# B&R Automation Studio project ControlPLC_DataDistribution
Automation Studio 4.11.3.51 SP; VulcanForms Printer Control PLC Gen 3.0; technology packages: mapp 5.19.0, mappCockpit 5.19.0, mappControl 5.19.0, mappMotion 5.19.3, mappSafety 5.19.0, mappView 5.19.0

## Configuration APC910

CPU 5PC900.TS17-02, AutomationRuntime D4.92, Build 4.1.2, Vc V4.72.5

### Hardware
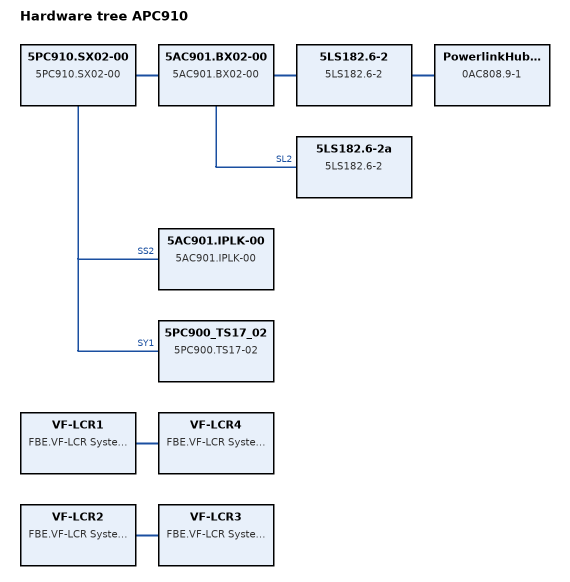
```
5AC901.BX02-00 : 5AC901.BX02-00 v1.0.1.0  [SY -> 5PC910.SX02-00.SY3]
5AC901.IPLK-00 : 5AC901.IPLK-00 v1.8.1.0  [SS -> 5PC910.SX02-00.SS2]
  Supervision = off
5LS182.6-2 : 5LS182.6-2 v1.9.0.0  [SL -> 5AC901.BX02-00.SL1]
  Connector IF1:
    CycleTime = 800
    EplNatSubnet = 192.168.102.0
  Supervision = off
5LS182.6-2a : 5LS182.6-2 v1.9.0.0  [SL -> 5AC901.BX02-00.SL2]
  Connector IF1:
    EplNatSubnet = 192.168.103.0
  Supervision = off
5PC900_TS17_02 : 5PC900.TS17-02 v2.1.0.0  [SY -> 5PC910.SX02-00.SY1]
  ConfigurationID = ControlPLC_LaserCleanroom_APC910
  UserPartitionSize = 5000
  UserRamDevice = PCI.2.LS182.SRAM
  UserRamSize = 1048320
  RemMemDevice = PCI.1.LS182.SRAM
  RemMemSize = 116736
  PermanentPvSize = 50000
  RemanentGlobalPvSize = 50000
  VolatileGlobalPvSize = 1100000
  ClearNvMemoryAfterShutdownFlushError = 0
  CyclicFlushRemMemSelector = 1
  RebootReset = 1
  FileDevice1
  FileDeviceName1 = USER
  FileDevicePath1 = USER_PATH
  FtpUser1
  FtpUsername1 = admin
  FtpUserPassword1 = cjYgzx2XKeawARoLvdaLrZty7HtHCNS4hNwff38YIhA=
  FtpUserSalt1 = Vifl6tjb
  FTPAccessRight1 = 0
  FTPdevice1 = ALL
  ActivateOpcUa = 1
  OpcUaPort = 4850
  OpcUa_Security_AdminRole = Administrators
  OpcUaLimitsMaxPublish = 50
  OpcUaInformationModels_PV_Version = 1
5PC910.SX02-00 : 5PC910.SX02-00 v2.1.2.0
  Connector IF1:
    AssignedOperatingSystem = ARemb
  Connector IF3:
    AssignedOperatingSystem = ARemb
    ActivateDevice = 1
    Mode = Manual
    InternetAddress = 192.168.200.50
    SubnetMask = 255.255.255.0
  Connector IF4:
    AssignedOperatingSystem = ARemb
    ActivateDevice = 1
  Connector IF5:
    AssignedOperatingSystem = ARemb
  Connector IF6:
    AssignedOperatingSystem = ARemb
  Connector IF7:
    AssignedOperatingSystem = ARemb
  Connector IF8:
    AssignedOperatingSystem = ARemb
  Connector IF9:
    AssignedOperatingSystem = ARemb
PowerlinkHub_DCEnclosure : 0AC808.9-1 v1.0.0.0  [ETH1 -> 5LS182.6-2.IF1 [Cable Type=PowerlinkCable, Length=10, Version=1.0.0.3]; ETH6 -> VF-LCR4.PLK2 [Cable Type=PowerlinkCable, Length=10, Version=1.0.0.3]]
VF-LCR1 : FBE.VF-LCR System (version 04) v04 (OrderNumber=VF-LCR)  [PLK1 -> VF-LCR2.PLK2 (NodeNumber=51) [Cable Type=PowerlinkCable, Length=10, Version=1.0.0.3]; PLK2 -> VF-LCR4.PLK1 (NodeNumber=51) [Cable Type=PowerlinkCable, Length=10, Version=1.0.0.3]]
  Supervision = off
  ResponseTimeout = 50
VF-LCR2 : FBE.VF-LCR System (version 04) v04 (OrderNumber=VF-LCR)  [PLK1 -> VF-LCR3.PLK2 (NodeNumber=52) [Cable Type=PowerlinkCable, Length=10, Version=1.0.0.3]; PLK2 -> VF-LCR1.PLK1 (NodeNumber=52) [Cable Type=PowerlinkCable, Length=10, Version=1.0.0.3]]
  Supervision = off
  ResponseTimeout = 50
VF-LCR3 : FBE.VF-LCR System (version 04) v04 (OrderNumber=VF-LCR)  [PLK2 -> VF-LCR2.PLK1 (NodeNumber=53) [Cable Type=PowerlinkCable, Length=10, Version=1.0.0.3]]
  Supervision = off
  ResponseTimeout = 50
VF-LCR4 : FBE.VF-LCR System (version 04) v04 (OrderNumber=VF-LCR)  [PLK1 -> VF-LCR1.PLK2 (NodeNumber=54) [Cable Type=PowerlinkCable, Length=10, Version=1.0.0.3]; PLK2 -> PowerlinkHub_DCEnclosure.ETH6 (NodeNumber=54) [Cable Type=PowerlinkCable, Length=10, Version=1.0.0.3]]
  Supervision = off
  ResponseTimeout = 50
```

### IoMap.iom - 5PC900_TS17_02/IoMap.iom
```iecst
VAR_CONFIG
	::VFLCR_Ope1:IO.raw.oSystemControl AT %QD."VF-LCR2".SYSTEM_CONTROL_I2004Out;
	::VFLCR_Ope1:IO.ao.SelectedPrintNumber AT %QD."VF-LCR2".SELECTED_PRINT_NUMBER_I200BOut;
	::VFLCR_Ope1:IO.ao.SelectedLayerNumber AT %QD."VF-LCR2".SELECTED_LAYER_NUMBER_I200COut;
	::VFLCR_Ope1:IO.ao.SelectedBuildLayout AT %QD."VF-LCR2".SELECTED_BUILD_LAYOUT_I200AOut;
	::VFLCR_Ope1:IO.ao.PLCHeartbeat AT %QD."VF-LCR2".PLC_HEARTBEAT_I2003Out;
	::VFLCR_Ope1:IO.raw.oOperationControl AT %QD."VF-LCR2".OPERATION_CONTROL_I2005Out;
	::VFLCR_Ope1:IO.raw.oManualLaserOperation AT %QD."VF-LCR2".MANUAL_LASER_OPERATION_I200EOut;
	::VFLCR_Ope1:IO.raw.oManualLaserCurrentSetpoint AT %QD."VF-LCR2".MANUAL_LASER_CURRENT_SETPOINT_I200FOut;
	::VFLCR_Ope1:IO.raw.oLaserEnable AT %QD."VF-LCR2".LASER_ENABLE_I2008Out;
	::VFLCR_Ope1:IO.raw.oEnableLaserMainPower AT %QD."VF-LCR2".LASER_REMOTE_START_I2010Out;
	::VFLCR_Ope1:IO.raw.oEnableLaserEmission AT %QD."VF-LCR2".LASER_EMISSION_CONTROL_I2012Out;
	::VFLCR_Ope1:IO.raw.oEnableGuideLaser AT %QD."VF-LCR2".GUIDE_LASER_CONTROL_I2011Out;
	::VFLCR_Ope1:IO.raw.oResetLaserErrors AT %QD."VF-LCR2".LASER_RESET_I2013Out;
	::VFLCR_Ope1:IO.di.PowerlinkModuleOK AT %IX."VF-LCR2".ModuleOk;
	::VFLCR_Ope1:IO.ai.DMACurrentTrajectory[0] AT %ID."VF-LCR2".Entry_I201B_S01;
	::VFLCR_Ope1:IO.raw.iLaserFatalError AT %ID."VF-LCR2".SYSTEM_ERROR_I2018;
	::VFLCR_Ope1:IO.raw.iSystemStatus AT %ID."VF-LCR2".SYSTEM_STATUS_I2006;
	::VFLCR_Ope1:IO.ai.SystemHeartbeat AT %ID."VF-LCR2".SYSTEM_HEARTBEAT_I2002;
	::VFLCR_Ope1:IO.raw.iSoftwareRevision AT %ID."VF-LCR2".SOFTWARE_REVISION_I201D;
	::VFLCR_Ope1:IO.raw.iOperationStatus AT %ID."VF-LCR2".OPERATION_STATUS_I2007;
	::VFLCR_Ope1:IO.raw.iManualModeLaserPower AT %ID."VF-LCR2".LASER_POWER_MONITOR_I2019;
	::VFLCR_Ope1:IO.ai.LUTFiles_CalibrationID AT %ID."VF-LCR2".LUT_LOAD_STATUS_I2009;
	::VFLCR_Ope1:IO.raw.iLaserWatchdogError AT %ID."VF-LCR2".LASER_WATCHDOG_ERROR_I201E;
	::VFLCR_Ope1:IO.raw.iLaserEmissionEnabled AT %ID."VF-LCR2".LASER_EMISSION_ON_I2017;
	::VFLCR_Ope1:IO.raw.iLaserControlPowerEnabled AT %ID."VF-LCR2".LASER_CONTROL_SYSTEM_POWERED_ON_I2015;
	::VFLCR_Ope1:IO.raw.iFPGARevision AT %ID."VF-LCR2".FPGA_REVISION_I2001;
	::VFLCR_Ope1:IO.ai.DMAStatus[8] AT %ID."VF-LCR2".Entry_I201A_S09;
	::VFLCR_Ope1:IO.ai.DMAStatus[7] AT %ID."VF-LCR2".Entry_I201A_S08;
	::VFLCR_Ope1:IO.ai.DMAStatus[6] AT %ID."VF-LCR2".Entry_I201A_S07;
	::VFLCR_Ope1:IO.ai.DMAStatus[5] AT %ID."VF-LCR2".Entry_I201A_S06;
	::VFLCR_Ope1:IO.ai.DMAStatus[4] AT %ID."VF-LCR2".Entry_I201A_S05;
	::VFLCR_Ope1:IO.ai.DMAStatus[3] AT %ID."VF-LCR2".Entry_I201A_S04;
	::VFLCR_Ope1:IO.ai.DMAStatus[13] AT %ID."VF-LCR2".Entry_I201A_S0E;
	::VFLCR_Ope1:IO.ai.DMAStatus[2] AT %ID."VF-LCR2".Entry_I201A_S03;
	::VFLCR_Ope1:IO.ai.DMAStatus[19] AT %ID."VF-LCR2".Entry_I201A_S14;
	::VFLCR_Ope1:IO.ai.DMAStatus[1] AT %ID."VF-LCR2".Entry_I201A_S02;
	::VFLCR_Ope1:IO.ai.DMAStatus[18] AT %ID."VF-LCR2".Entry_I201A_S13;
	::VFLCR_Ope1:IO.ai.DMAStatus[17] AT %ID."VF-LCR2".Entry_I201A_S12;
	::VFLCR_Ope1:IO.ai.DMAStatus[16] AT %ID."VF-LCR2".Entry_I201A_S11;
	::VFLCR_Ope1:IO.ai.DMAStatus[15] AT %ID."VF-LCR2".Entry_I201A_S10;
	::VFLCR_Ope1:IO.ai.DMAStatus[14] AT %ID."VF-LCR2".Entry_I201A_S0F;
	::VFLCR_Ope1:IO.raw.iLaserMainPowerEnabled AT %ID."VF-LCR2".LASER_MAIN_POWER_ON_I2016;
	::VFLCR_Ope1:IO.raw.iLaserReady_Error AT %ID."VF-LCR2".LASER_ERROR_READY_I2014;
	::VFLCR_Ope1:IO.ai.DMAStatus[20] AT %ID."VF-LCR2".Entry_I201A_S15;
	::VFLCR_Ope1:IO.ai.DMAStatus[12] AT %ID."VF-LCR2".Entry_I201A_S0D;
	::VFLCR_Ope1:IO.ai.DMACurrentTrajectory[7] AT %ID."VF-LCR2".Entry_I201B_S08;
	::VFLCR_Ope1:IO.ai.DMAStatus[0] AT %ID."VF-LCR2".Entry_I201A_S01;
	::VFLCR_Ope1:IO.ai.DMALastPacketPosition[8] AT %ID."VF-LCR2".Entry_I201C_S09;
	::VFLCR_Ope1:IO.ai.DMALastPacketPosition[7] AT %ID."VF-LCR2".Entry_I201C_S08;
	::VFLCR_Ope1:IO.ai.DMALastPacketPosition[6] AT %ID."VF-LCR2".Entry_I201C_S07;
	::VFLCR_Ope1:IO.ai.DMALastPacketPosition[5] AT %ID."VF-LCR2".Entry_I201C_S06;
	::VFLCR_Ope1:IO.ai.DMALastPacketPosition[4] AT %ID."VF-LCR2".Entry_I201C_S05;
	::VFLCR_Ope1:IO.ai.DMALastPacketPosition[3] AT %ID."VF-LCR2".Entry_I201C_S04;
	::VFLCR_Ope1:IO.ai.DMALastPacketPosition[2] AT %ID."VF-LCR2".Entry_I201C_S03;
	::VFLCR_Ope1:IO.ai.DMALastPacketPosition[19] AT %ID."VF-LCR2".Entry_I201C_S14;
	::VFLCR_Ope1:IO.ai.DMAStatus[9] AT %ID."VF-LCR2".Entry_I201A_S0A;
	::VFLCR_Ope1:IO.ai.DMALastPacketPosition[20] AT %ID."VF-LCR2".Entry_I201C_S15;
	::VFLCR_Ope1:IO.ai.DMALastPacketPosition[18] AT %ID."VF-LCR2".Entry_I201C_S13;
	::VFLCR_Ope1:IO.ai.DMALastPacketPosition[17] AT %ID."VF-LCR2".Entry_I201C_S12;
	::VFLCR_Ope1:IO.ai.DMALastPacketPosition[16] AT %ID."VF-LCR2".Entry_I201C_S11;
	::VFLCR_Ope1:IO.ai.DMALastPacketPosition[15] AT %ID."VF-LCR2".Entry_I201C_S10;
	::VFLCR_Ope1:IO.ai.DMALastPacketPosition[14] AT %ID."VF-LCR2".Entry_I201C_S0F;
	::VFLCR_Ope1:IO.ai.DMALastPacketPosition[13] AT %ID."VF-LCR2".Entry_I201C_S0E;
	::VFLCR_Ope1:IO.ai.DMALastPacketPosition[12] AT %ID."VF-LCR2".Entry_I201C_S0D;
	::VFLCR_Ope1:IO.ai.DMALastPacketPosition[11] AT %ID."VF-LCR2".Entry_I201C_S0C;
	::VFLCR_Ope1:IO.ai.DMAStatus[10] AT %ID."VF-LCR2".Entry_I201A_S0B;
	::VFLCR_Ope1:IO.ai.DMALastPacketPosition[1] AT %ID."VF-LCR2".Entry_I201C_S02;
	::VFLCR_Ope1:IO.ai.DMAStatus[11] AT %ID."VF-LCR2".Entry_I201A_S0C;
	::VFLCR_Ope1:IO.ai.DMALastPacketPosition[10] AT %ID."VF-LCR2".Entry_I201C_S0B;
	::VFLCR_Ope1:IO.ai.DMALastPacketPosition[0] AT %ID."VF-LCR2".Entry_I201C_S01;
	::VFLCR_Ope1:IO.ai.DMACurrentTrajectory[6] AT %ID."VF-LCR2".Entry_I201B_S07;
	::VFLCR_Ope1:IO.ai.DMACurrentTrajectory[5] AT %ID."VF-LCR2".Entry_I201B_S06;
	::VFLCR_Ope1:IO.ai.DMACurrentTrajectory[4] AT %ID."VF-LCR2".Entry_I201B_S05;
	::VFLCR_Ope1:IO.ai.DMACurrentTrajectory[3] AT %ID."VF-LCR2".Entry_I201B_S04;
	::VFLCR_Ope1:IO.ai.DMACurrentTrajectory[2] AT %ID."VF-LCR2".Entry_I201B_S03;
	::VFLCR_Ope1:IO.ai.DMACurrentTrajectory[20] AT %ID."VF-LCR2".Entry_I201B_S15;
	::VFLCR_Ope1:IO.ai.DMACurrentTrajectory[19] AT %ID."VF-LCR2".Entry_I201B_S14;
	::VFLCR_Ope1:IO.ai.DMACurrentTrajectory[1] AT %ID."VF-LCR2".Entry_I201B_S02;
	::VFLCR_Ope1:IO.ai.DMACurrentTrajectory[18] AT %ID."VF-LCR2".Entry_I201B_S13;
	::VFLCR_Ope1:IO.ai.DMALastPacketPosition[9] AT %ID."VF-LCR2".Entry_I201C_S0A;
	::VFLCR_Ope1:IO.ai.DMACurrentTrajectory[17] AT %ID."VF-LCR2".Entry_I201B_S12;
	::VFLCR_Ope1:IO.ai.DMACurrentTrajectory[15] AT %ID."VF-LCR2".Entry_I201B_S10;
	::VFLCR_Ope1:IO.ai.DMACurrentTrajectory[14] AT %ID."VF-LCR2".Entry_I201B_S0F;
	::VFLCR_Ope1:IO.ai.DMACurrentTrajectory[13] AT %ID."VF-LCR2".Entry_I201B_S0E;
	::VFLCR_Ope1:IO.ai.DMACurrentTrajectory[12] AT %ID."VF-LCR2".Entry_I201B_S0D;
	::VFLCR_Ope1:IO.ai.DMACurrentTrajectory[11] AT %ID."VF-LCR2".Entry_I201B_S0C;
	::VFLCR_Ope1:IO.ai.DMACurrentTrajectory[10] AT %ID."VF-LCR2".Entry_I201B_S0B;
	::VFLCR_Ope1:IO.ai.DMACurrentTrajectory[9] AT %ID."VF-LCR2".Entry_I201B_S0A;
	::VFLCR_Ope1:IO.ai.DMACurrentTrajectory[8] AT %ID."VF-LCR2".Entry_I201B_S09;
	::VFLCR_Ope1:IO.ai.DMACurrentTrajectory[16] AT %ID."VF-LCR2".Entry_I201B_S11;
	::VFLCR_Ope2:IO.raw.oSystemControl AT %QD."VF-LCR3".SYSTEM_CONTROL_I2004Out;
	::VFLCR_Ope2:IO.ao.SelectedPrintNumber AT %QD."VF-LCR3".SELECTED_PRINT_NUMBER_I200BOut;
	::VFLCR_Ope2:IO.ao.SelectedLayerNumber AT %QD."VF-LCR3".SELECTED_LAYER_NUMBER_I200COut;
	::VFLCR_Ope2:IO.ao.SelectedBuildLayout AT %QD."VF-LCR3".SELECTED_BUILD_LAYOUT_I200AOut;
	::VFLCR_Ope2:IO.ao.PLCHeartbeat AT %QD."VF-LCR3".PLC_HEARTBEAT_I2003Out;
	::VFLCR_Ope2:IO.raw.oOperationControl AT %QD."VF-LCR3".OPERATION_CONTROL_I2005Out;
	::VFLCR_Ope2:IO.raw.oManualLaserOperation AT %QD."VF-LCR3".MANUAL_LASER_OPERATION_I200EOut;
	::VFLCR_Ope2:IO.raw.oManualLaserCurrentSetpoint AT %QD."VF-LCR3".MANUAL_LASER_CURRENT_SETPOINT_I200FOut;
	::VFLCR_Ope2:IO.raw.oLaserEnable AT %QD."VF-LCR3".LASER_ENABLE_I2008Out;
	::VFLCR_Ope2:IO.raw.oEnableLaserMainPower AT %QD."VF-LCR3".LASER_REMOTE_START_I2010Out;
	::VFLCR_Ope2:IO.raw.oEnableLaserEmission AT %QD."VF-LCR3".LASER_EMISSION_CONTROL_I2012Out;
	::VFLCR_Ope2:IO.raw.oEnableGuideLaser AT %QD."VF-LCR3".GUIDE_LASER_CONTROL_I2011Out;
	::VFLCR_Ope2:IO.raw.oResetLaserErrors AT %QD."VF-LCR3".LASER_RESET_I2013Out;
	::VFLCR_Ope2:IO.di.PowerlinkModuleOK AT %IX."VF-LCR3".ModuleOk;
	::VFLCR_Ope2:IO.ai.DMACurrentTrajectory[0] AT %ID."VF-LCR3".Entry_I201B_S01;
	::VFLCR_Ope2:IO.raw.iLaserFatalError AT %ID."VF-LCR3".SYSTEM_ERROR_I2018;
	::VFLCR_Ope2:IO.raw.iSystemStatus AT %ID."VF-LCR3".SYSTEM_STATUS_I2006;
	::VFLCR_Ope2:IO.ai.SystemHeartbeat AT %ID."VF-LCR3".SYSTEM_HEARTBEAT_I2002;
	::VFLCR_Ope2:IO.raw.iSoftwareRevision AT %ID."VF-LCR3".SOFTWARE_REVISION_I201D;
	::VFLCR_Ope2:IO.raw.iOperationStatus AT %ID."VF-LCR3".OPERATION_STATUS_I2007;
	::VFLCR_Ope2:IO.raw.iManualModeLaserPower AT %ID."VF-LCR3".LASER_POWER_MONITOR_I2019;
	::VFLCR_Ope2:IO.ai.LUTFiles_CalibrationID AT %ID."VF-LCR3".LUT_LOAD_STATUS_I2009;
	::VFLCR_Ope2:IO.raw.iLaserWatchdogError AT %ID."VF-LCR3".LASER_WATCHDOG_ERROR_I201E;
	::VFLCR_Ope2:IO.raw.iLaserEmissionEnabled AT %ID."VF-LCR3".LASER_EMISSION_ON_I2017;
	::VFLCR_Ope2:IO.raw.iLaserControlPowerEnabled AT %ID."VF-LCR3".LASER_CONTROL_SYSTEM_POWERED_ON_I2015;
	::VFLCR_Ope2:IO.raw.iFPGARevision AT %ID."VF-LCR3".FPGA_REVISION_I2001;
	::VFLCR_Ope2:IO.ai.DMAStatus[8] AT %ID."VF-LCR3".Entry_I201A_S09;
	::VFLCR_Ope2:IO.ai.DMAStatus[7] AT %ID."VF-LCR3".Entry_I201A_S08;
	::VFLCR_Ope2:IO.ai.DMAStatus[6] AT %ID."VF-LCR3".Entry_I201A_S07;
	::VFLCR_Ope2:IO.ai.DMAStatus[5] AT %ID."VF-LCR3".Entry_I201A_S06;
	::VFLCR_Ope2:IO.ai.DMAStatus[4] AT %ID."VF-LCR3".Entry_I201A_S05;
	::VFLCR_Ope2:IO.ai.DMAStatus[3] AT %ID."VF-LCR3".Entry_I201A_S04;
	::VFLCR_Ope2:IO.ai.DMAStatus[13] AT %ID."VF-LCR3".Entry_I201A_S0E;
	::VFLCR_Ope2:IO.ai.DMAStatus[2] AT %ID."VF-LCR3".Entry_I201A_S03;
	::VFLCR_Ope2:IO.ai.DMAStatus[19] AT %ID."VF-LCR3".Entry_I201A_S14;
	::VFLCR_Ope2:IO.ai.DMAStatus[1] AT %ID."VF-LCR3".Entry_I201A_S02;
	::VFLCR_Ope2:IO.ai.DMAStatus[18] AT %ID."VF-LCR3".Entry_I201A_S13;
	::VFLCR_Ope2:IO.ai.DMAStatus[17] AT %ID."VF-LCR3".Entry_I201A_S12;
	::VFLCR_Ope2:IO.ai.DMAStatus[16] AT %ID."VF-LCR3".Entry_I201A_S11;
	::VFLCR_Ope2:IO.ai.DMAStatus[15] AT %ID."VF-LCR3".Entry_I201A_S10;
	::VFLCR_Ope2:IO.ai.DMAStatus[14] AT %ID."VF-LCR3".Entry_I201A_S0F;
	::VFLCR_Ope2:IO.raw.iLaserMainPowerEnabled AT %ID."VF-LCR3".LASER_MAIN_POWER_ON_I2016;
	::VFLCR_Ope2:IO.raw.iLaserReady_Error AT %ID."VF-LCR3".LASER_ERROR_READY_I2014;
	::VFLCR_Ope2:IO.ai.DMAStatus[20] AT %ID."VF-LCR3".Entry_I201A_S15;
	::VFLCR_Ope2:IO.ai.DMAStatus[12] AT %ID."VF-LCR3".Entry_I201A_S0D;
	::VFLCR_Ope2:IO.ai.DMACurrentTrajectory[7] AT %ID."VF-LCR3".Entry_I201B_S08;
	::VFLCR_Ope2:IO.ai.DMAStatus[0] AT %ID."VF-LCR3".Entry_I201A_S01;
	::VFLCR_Ope2:IO.ai.DMALastPacketPosition[8] AT %ID."VF-LCR3".Entry_I201C_S09;
	::VFLCR_Ope2:IO.ai.DMALastPacketPosition[7] AT %ID."VF-LCR3".Entry_I201C_S08;
	::VFLCR_Ope2:IO.ai.DMALastPacketPosition[6] AT %ID."VF-LCR3".Entry_I201C_S07;
	::VFLCR_Ope2:IO.ai.DMALastPacketPosition[5] AT %ID."VF-LCR3".Entry_I201C_S06;
	::VFLCR_Ope2:IO.ai.DMALastPacketPosition[4] AT %ID."VF-LCR3".Entry_I201C_S05;
	::VFLCR_Ope2:IO.ai.DMALastPacketPosition[3] AT %ID."VF-LCR3".Entry_I201C_S04;
	::VFLCR_Ope2:IO.ai.DMALastPacketPosition[2] AT %ID."VF-LCR3".Entry_I201C_S03;
	::VFLCR_Ope2:IO.ai.DMALastPacketPosition[19] AT %ID."VF-LCR3".Entry_I201C_S14;
	::VFLCR_Ope2:IO.ai.DMAStatus[9] AT %ID."VF-LCR3".Entry_I201A_S0A;
	::VFLCR_Ope2:IO.ai.DMALastPacketPosition[20] AT %ID."VF-LCR3".Entry_I201C_S15;
	::VFLCR_Ope2:IO.ai.DMALastPacketPosition[18] AT %ID."VF-LCR3".Entry_I201C_S13;
	::VFLCR_Ope2:IO.ai.DMALastPacketPosition[17] AT %ID."VF-LCR3".Entry_I201C_S12;
	::VFLCR_Ope2:IO.ai.DMALastPacketPosition[16] AT %ID."VF-LCR3".Entry_I201C_S11;
	::VFLCR_Ope2:IO.ai.DMALastPacketPosition[15] AT %ID."VF-LCR3".Entry_I201C_S10;
	::VFLCR_Ope2:IO.ai.DMALastPacketPosition[14] AT %ID."VF-LCR3".Entry_I201C_S0F;
	::VFLCR_Ope2:IO.ai.DMALastPacketPosition[13] AT %ID."VF-LCR3".Entry_I201C_S0E;
	::VFLCR_Ope2:IO.ai.DMALastPacketPosition[12] AT %ID."VF-LCR3".Entry_I201C_S0D;
	::VFLCR_Ope2:IO.ai.DMALastPacketPosition[11] AT %ID."VF-LCR3".Entry_I201C_S0C;
	::VFLCR_Ope2:IO.ai.DMAStatus[10] AT %ID."VF-LCR3".Entry_I201A_S0B;
	::VFLCR_Ope2:IO.ai.DMALastPacketPosition[1] AT %ID."VF-LCR3".Entry_I201C_S02;
	::VFLCR_Ope2:IO.ai.DMAStatus[11] AT %ID."VF-LCR3".Entry_I201A_S0C;
	::VFLCR_Ope2:IO.ai.DMALastPacketPosition[10] AT %ID."VF-LCR3".Entry_I201C_S0B;
	::VFLCR_Ope2:IO.ai.DMALastPacketPosition[0] AT %ID."VF-LCR3".Entry_I201C_S01;
	::VFLCR_Ope2:IO.ai.DMACurrentTrajectory[6] AT %ID."VF-LCR3".Entry_I201B_S07;
	::VFLCR_Ope2:IO.ai.DMACurrentTrajectory[5] AT %ID."VF-LCR3".Entry_I201B_S06;
	::VFLCR_Ope2:IO.ai.DMACurrentTrajectory[4] AT %ID."VF-LCR3".Entry_I201B_S05;
	::VFLCR_Ope2:IO.ai.DMACurrentTrajectory[3] AT %ID."VF-LCR3".Entry_I201B_S04;
	::VFLCR_Ope2:IO.ai.DMACurrentTrajectory[2] AT %ID."VF-LCR3".Entry_I201B_S03;
	::VFLCR_Ope2:IO.ai.DMACurrentTrajectory[20] AT %ID."VF-LCR3".Entry_I201B_S15;
	::VFLCR_Ope2:IO.ai.DMACurrentTrajectory[19] AT %ID."VF-LCR3".Entry_I201B_S14;
	::VFLCR_Ope2:IO.ai.DMACurrentTrajectory[1] AT %ID."VF-LCR3".Entry_I201B_S02;
	::VFLCR_Ope2:IO.ai.DMACurrentTrajectory[18] AT %ID."VF-LCR3".Entry_I201B_S13;
	::VFLCR_Ope2:IO.ai.DMALastPacketPosition[9] AT %ID."VF-LCR3".Entry_I201C_S0A;
	::VFLCR_Ope2:IO.ai.DMACurrentTrajectory[17] AT %ID."VF-LCR3".Entry_I201B_S12;
	::VFLCR_Ope2:IO.ai.DMACurrentTrajectory[15] AT %ID."VF-LCR3".Entry_I201B_S10;
	::VFLCR_Ope2:IO.ai.DMACurrentTrajectory[14] AT %ID."VF-LCR3".Entry_I201B_S0F;
	::VFLCR_Ope2:IO.ai.DMACurrentTrajectory[13] AT %ID."VF-LCR3".Entry_I201B_S0E;
	::VFLCR_Ope2:IO.ai.DMACurrentTrajectory[12] AT %ID."VF-LCR3".Entry_I201B_S0D;
	::VFLCR_Ope2:IO.ai.DMACurrentTrajectory[11] AT %ID."VF-LCR3".Entry_I201B_S0C;
	::VFLCR_Ope2:IO.ai.DMACurrentTrajectory[10] AT %ID."VF-LCR3".Entry_I201B_S0B;
	::VFLCR_Ope2:IO.ai.DMACurrentTrajectory[9] AT %ID."VF-LCR3".Entry_I201B_S0A;
	::VFLCR_Ope2:IO.ai.DMACurrentTrajectory[8] AT %ID."VF-LCR3".Entry_I201B_S09;
	::VFLCR_Ope2:IO.ai.DMACurrentTrajectory[16] AT %ID."VF-LCR3".Entry_I201B_S11;
	::VFLCR_Ope3:IO.raw.oSystemControl AT %QD."VF-LCR4".SYSTEM_CONTROL_I2004Out;
	::VFLCR_Ope3:IO.ao.SelectedPrintNumber AT %QD."VF-LCR4".SELECTED_PRINT_NUMBER_I200BOut;
	::VFLCR_Ope3:IO.ao.SelectedLayerNumber AT %QD."VF-LCR4".SELECTED_LAYER_NUMBER_I200COut;
	::VFLCR_Ope3:IO.ao.SelectedBuildLayout AT %QD."VF-LCR4".SELECTED_BUILD_LAYOUT_I200AOut;
	::VFLCR_Ope3:IO.ao.PLCHeartbeat AT %QD."VF-LCR4".PLC_HEARTBEAT_I2003Out;
	::VFLCR_Ope3:IO.raw.oOperationControl AT %QD."VF-LCR4".OPERATION_CONTROL_I2005Out;
	::VFLCR_Ope3:IO.raw.oManualLaserOperation AT %QD."VF-LCR4".MANUAL_LASER_OPERATION_I200EOut;
	::VFLCR_Ope3:IO.raw.oManualLaserCurrentSetpoint AT %QD."VF-LCR4".MANUAL_LASER_CURRENT_SETPOINT_I200FOut;
	::VFLCR_Ope3:IO.raw.oLaserEnable AT %QD."VF-LCR4".LASER_ENABLE_I2008Out;
	::VFLCR_Ope3:IO.raw.oEnableLaserMainPower AT %QD."VF-LCR4".LASER_REMOTE_START_I2010Out;
	::VFLCR_Ope3:IO.raw.oEnableLaserEmission AT %QD."VF-LCR4".LASER_EMISSION_CONTROL_I2012Out;
	::VFLCR_Ope3:IO.raw.oEnableGuideLaser AT %QD."VF-LCR4".GUIDE_LASER_CONTROL_I2011Out;
	::VFLCR_Ope3:IO.raw.oResetLaserErrors AT %QD."VF-LCR4".LASER_RESET_I2013Out;
	::VFLCR_Ope3:IO.di.PowerlinkModuleOK AT %IX."VF-LCR4".ModuleOk;
	::VFLCR_Ope3:IO.ai.DMACurrentTrajectory[0] AT %ID."VF-LCR4".Entry_I201B_S01;
	::VFLCR_Ope3:IO.raw.iLaserFatalError AT %ID."VF-LCR4".SYSTEM_ERROR_I2018;
	::VFLCR_Ope3:IO.raw.iSystemStatus AT %ID."VF-LCR4".SYSTEM_STATUS_I2006;
	::VFLCR_Ope3:IO.ai.SystemHeartbeat AT %ID."VF-LCR4".SYSTEM_HEARTBEAT_I2002;
	::VFLCR_Ope3:IO.raw.iSoftwareRevision AT %ID."VF-LCR4".SOFTWARE_REVISION_I201D;
	::VFLCR_Ope3:IO.raw.iOperationStatus AT %ID."VF-LCR4".OPERATION_STATUS_I2007;
	::VFLCR_Ope3:IO.raw.iManualModeLaserPower AT %ID."VF-LCR4".LASER_POWER_MONITOR_I2019;
	::VFLCR_Ope3:IO.ai.LUTFiles_CalibrationID AT %ID."VF-LCR4".LUT_LOAD_STATUS_I2009;
	::VFLCR_Ope3:IO.raw.iLaserWatchdogError AT %ID."VF-LCR4".LASER_WATCHDOG_ERROR_I201E;
	::VFLCR_Ope3:IO.raw.iLaserEmissionEnabled AT %ID."VF-LCR4".LASER_EMISSION_ON_I2017;
	::VFLCR_Ope3:IO.raw.iLaserControlPowerEnabled AT %ID."VF-LCR4".LASER_CONTROL_SYSTEM_POWERED_ON_I2015;
	::VFLCR_Ope3:IO.raw.iFPGARevision AT %ID."VF-LCR4".FPGA_REVISION_I2001;
	::VFLCR_Ope3:IO.ai.DMAStatus[8] AT %ID."VF-LCR4".Entry_I201A_S09;
	::VFLCR_Ope3:IO.ai.DMAStatus[7] AT %ID."VF-LCR4".Entry_I201A_S08;
	::VFLCR_Ope3:IO.ai.DMAStatus[6] AT %ID."VF-LCR4".Entry_I201A_S07;
	::VFLCR_Ope3:IO.ai.DMAStatus[5] AT %ID."VF-LCR4".Entry_I201A_S06;
	::VFLCR_Ope3:IO.ai.DMAStatus[4] AT %ID."VF-LCR4".Entry_I201A_S05;
	::VFLCR_Ope3:IO.ai.DMAStatus[3] AT %ID."VF-LCR4".Entry_I201A_S04;
	::VFLCR_Ope3:IO.ai.DMAStatus[13] AT %ID."VF-LCR4".Entry_I201A_S0E;
	::VFLCR_Ope3:IO.ai.DMAStatus[2] AT %ID."VF-LCR4".Entry_I201A_S03;
	::VFLCR_Ope3:IO.ai.DMAStatus[19] AT %ID."VF-LCR4".Entry_I201A_S14;
	::VFLCR_Ope3:IO.ai.DMAStatus[1] AT %ID."VF-LCR4".Entry_I201A_S02;
	::VFLCR_Ope3:IO.ai.DMAStatus[18] AT %ID."VF-LCR4".Entry_I201A_S13;
	::VFLCR_Ope3:IO.ai.DMAStatus[17] AT %ID."VF-LCR4".Entry_I201A_S12;
	::VFLCR_Ope3:IO.ai.DMAStatus[16] AT %ID."VF-LCR4".Entry_I201A_S11;
	::VFLCR_Ope3:IO.ai.DMAStatus[15] AT %ID."VF-LCR4".Entry_I201A_S10;
	::VFLCR_Ope3:IO.ai.DMAStatus[14] AT %ID."VF-LCR4".Entry_I201A_S0F;
	::VFLCR_Ope3:IO.raw.iLaserMainPowerEnabled AT %ID."VF-LCR4".LASER_MAIN_POWER_ON_I2016;
	::VFLCR_Ope3:IO.raw.iLaserReady_Error AT %ID."VF-LCR4".LASER_ERROR_READY_I2014;
	::VFLCR_Ope3:IO.ai.DMAStatus[20] AT %ID."VF-LCR4".Entry_I201A_S15;
	::VFLCR_Ope3:IO.ai.DMAStatus[12] AT %ID."VF-LCR4".Entry_I201A_S0D;
	::VFLCR_Ope3:IO.ai.DMACurrentTrajectory[7] AT %ID."VF-LCR4".Entry_I201B_S08;
	::VFLCR_Ope3:IO.ai.DMAStatus[0] AT %ID."VF-LCR4".Entry_I201A_S01;
	::VFLCR_Ope3:IO.ai.DMALastPacketPosition[8] AT %ID."VF-LCR4".Entry_I201C_S09;
	::VFLCR_Ope3:IO.ai.DMALastPacketPosition[7] AT %ID."VF-LCR4".Entry_I201C_S08;
	::VFLCR_Ope3:IO.ai.DMALastPacketPosition[6] AT %ID."VF-LCR4".Entry_I201C_S07;
	::VFLCR_Ope3:IO.ai.DMALastPacketPosition[5] AT %ID."VF-LCR4".Entry_I201C_S06;
	::VFLCR_Ope3:IO.ai.DMALastPacketPosition[4] AT %ID."VF-LCR4".Entry_I201C_S05;
	::VFLCR_Ope3:IO.ai.DMALastPacketPosition[3] AT %ID."VF-LCR4".Entry_I201C_S04;
	::VFLCR_Ope3:IO.ai.DMALastPacketPosition[2] AT %ID."VF-LCR4".Entry_I201C_S03;
	::VFLCR_Ope3:IO.ai.DMALastPacketPosition[19] AT %ID."VF-LCR4".Entry_I201C_S14;
	::VFLCR_Ope3:IO.ai.DMAStatus[9] AT %ID."VF-LCR4".Entry_I201A_S0A;
	::VFLCR_Ope3:IO.ai.DMALastPacketPosition[20] AT %ID."VF-LCR4".Entry_I201C_S15;
	::VFLCR_Ope3:IO.ai.DMALastPacketPosition[18] AT %ID."VF-LCR4".Entry_I201C_S13;
	::VFLCR_Ope3:IO.ai.DMALastPacketPosition[17] AT %ID."VF-LCR4".Entry_I201C_S12;
	::VFLCR_Ope3:IO.ai.DMALastPacketPosition[16] AT %ID."VF-LCR4".Entry_I201C_S11;
	::VFLCR_Ope3:IO.ai.DMALastPacketPosition[15] AT %ID."VF-LCR4".Entry_I201C_S10;
	::VFLCR_Ope3:IO.ai.DMALastPacketPosition[14] AT %ID."VF-LCR4".Entry_I201C_S0F;
	::VFLCR_Ope3:IO.ai.DMALastPacketPosition[13] AT %ID."VF-LCR4".Entry_I201C_S0E;
	::VFLCR_Ope3:IO.ai.DMALastPacketPosition[12] AT %ID."VF-LCR4".Entry_I201C_S0D;
	::VFLCR_Ope3:IO.ai.DMALastPacketPosition[11] AT %ID."VF-LCR4".Entry_I201C_S0C;
	::VFLCR_Ope3:IO.ai.DMAStatus[10] AT %ID."VF-LCR4".Entry_I201A_S0B;
	::VFLCR_Ope3:IO.ai.DMALastPacketPosition[1] AT %ID."VF-LCR4".Entry_I201C_S02;
	::VFLCR_Ope3:IO.ai.DMAStatus[11] AT %ID."VF-LCR4".Entry_I201A_S0C;
	::VFLCR_Ope3:IO.ai.DMALastPacketPosition[10] AT %ID."VF-LCR4".Entry_I201C_S0B;
	::VFLCR_Ope3:IO.ai.DMALastPacketPosition[0] AT %ID."VF-LCR4".Entry_I201C_S01;
	::VFLCR_Ope3:IO.ai.DMACurrentTrajectory[6] AT %ID."VF-LCR4".Entry_I201B_S07;
	::VFLCR_Ope3:IO.ai.DMACurrentTrajectory[5] AT %ID."VF-LCR4".Entry_I201B_S06;
	::VFLCR_Ope3:IO.ai.DMACurrentTrajectory[4] AT %ID."VF-LCR4".Entry_I201B_S05;
	::VFLCR_Ope3:IO.ai.DMACurrentTrajectory[3] AT %ID."VF-LCR4".Entry_I201B_S04;
	::VFLCR_Ope3:IO.ai.DMACurrentTrajectory[2] AT %ID."VF-LCR4".Entry_I201B_S03;
	::VFLCR_Ope3:IO.ai.DMACurrentTrajectory[20] AT %ID."VF-LCR4".Entry_I201B_S15;
	::VFLCR_Ope3:IO.ai.DMACurrentTrajectory[19] AT %ID."VF-LCR4".Entry_I201B_S14;
	::VFLCR_Ope3:IO.ai.DMACurrentTrajectory[1] AT %ID."VF-LCR4".Entry_I201B_S02;
	::VFLCR_Ope3:IO.ai.DMACurrentTrajectory[18] AT %ID."VF-LCR4".Entry_I201B_S13;
	::VFLCR_Ope3:IO.ai.DMALastPacketPosition[9] AT %ID."VF-LCR4".Entry_I201C_S0A;
	::VFLCR_Ope3:IO.ai.DMACurrentTrajectory[17] AT %ID."VF-LCR4".Entry_I201B_S12;
	::VFLCR_Ope3:IO.ai.DMACurrentTrajectory[15] AT %ID."VF-LCR4".Entry_I201B_S10;
	::VFLCR_Ope3:IO.ai.DMACurrentTrajectory[14] AT %ID."VF-LCR4".Entry_I201B_S0F;
	::VFLCR_Ope3:IO.ai.DMACurrentTrajectory[13] AT %ID."VF-LCR4".Entry_I201B_S0E;
	::VFLCR_Ope3:IO.ai.DMACurrentTrajectory[12] AT %ID."VF-LCR4".Entry_I201B_S0D;
	::VFLCR_Ope3:IO.ai.DMACurrentTrajectory[11] AT %ID."VF-LCR4".Entry_I201B_S0C;
	::VFLCR_Ope3:IO.ai.DMACurrentTrajectory[10] AT %ID."VF-LCR4".Entry_I201B_S0B;
	::VFLCR_Ope3:IO.ai.DMACurrentTrajectory[9] AT %ID."VF-LCR4".Entry_I201B_S0A;
	::VFLCR_Ope3:IO.ai.DMACurrentTrajectory[8] AT %ID."VF-LCR4".Entry_I201B_S09;
	::VFLCR_Ope3:IO.ai.DMACurrentTrajectory[16] AT %ID."VF-LCR4".Entry_I201B_S11;
	::VFLCR_Ope0:IO.raw.oSystemControl AT %QD."VF-LCR1".SYSTEM_CONTROL_I2004Out;
	::VFLCR_Ope0:IO.ao.SelectedPrintNumber AT %QD."VF-LCR1".SELECTED_PRINT_NUMBER_I200BOut;
	::VFLCR_Ope0:IO.ao.SelectedLayerNumber AT %QD."VF-LCR1".SELECTED_LAYER_NUMBER_I200COut;
	::VFLCR_Ope0:IO.ao.SelectedBuildLayout AT %QD."VF-LCR1".SELECTED_BUILD_LAYOUT_I200AOut;
	::VFLCR_Ope0:IO.ao.PLCHeartbeat AT %QD."VF-LCR1".PLC_HEARTBEAT_I2003Out;
	::VFLCR_Ope0:IO.raw.oOperationControl AT %QD."VF-LCR1".OPERATION_CONTROL_I2005Out;
	::VFLCR_Ope0:IO.raw.oManualLaserOperation AT %QD."VF-LCR1".MANUAL_LASER_OPERATION_I200EOut;
	::VFLCR_Ope0:IO.raw.oManualLaserCurrentSetpoint AT %QD."VF-LCR1".MANUAL_LASER_CURRENT_SETPOINT_I200FOut;
	::VFLCR_Ope0:IO.raw.oLaserEnable AT %QD."VF-LCR1".LASER_ENABLE_I2008Out;
	::VFLCR_Ope0:IO.raw.oEnableLaserMainPower AT %QD."VF-LCR1".LASER_REMOTE_START_I2010Out;
	::VFLCR_Ope0:IO.raw.oEnableLaserEmission AT %QD."VF-LCR1".LASER_EMISSION_CONTROL_I2012Out;
	::VFLCR_Ope0:IO.raw.oEnableGuideLaser AT %QD."VF-LCR1".GUIDE_LASER_CONTROL_I2011Out;
	::VFLCR_Ope0:IO.raw.oResetLaserErrors AT %QD."VF-LCR1".LASER_RESET_I2013Out;
	::VFLCR_Ope0:IO.di.PowerlinkModuleOK AT %IX."VF-LCR1".ModuleOk;
	::VFLCR_Ope0:IO.ai.DMACurrentTrajectory[0] AT %ID."VF-LCR1".Entry_I201B_S01;
	::VFLCR_Ope0:IO.raw.iLaserFatalError AT %ID."VF-LCR1".SYSTEM_ERROR_I2018;
	::VFLCR_Ope0:IO.raw.iSystemStatus AT %ID."VF-LCR1".SYSTEM_STATUS_I2006;
	::VFLCR_Ope0:IO.ai.SystemHeartbeat AT %ID."VF-LCR1".SYSTEM_HEARTBEAT_I2002;
	::VFLCR_Ope0:IO.raw.iSoftwareRevision AT %ID."VF-LCR1".SOFTWARE_REVISION_I201D;
	::VFLCR_Ope0:IO.raw.iOperationStatus AT %ID."VF-LCR1".OPERATION_STATUS_I2007;
	::VFLCR_Ope0:IO.raw.iManualModeLaserPower AT %ID."VF-LCR1".LASER_POWER_MONITOR_I2019;
	::VFLCR_Ope0:IO.ai.LUTFiles_CalibrationID AT %ID."VF-LCR1".LUT_LOAD_STATUS_I2009;
	::VFLCR_Ope0:IO.raw.iLaserWatchdogError AT %ID."VF-LCR1".LASER_WATCHDOG_ERROR_I201E;
	::VFLCR_Ope0:IO.raw.iLaserEmissionEnabled AT %ID."VF-LCR1".LASER_EMISSION_ON_I2017;
	::VFLCR_Ope0:IO.raw.iLaserControlPowerEnabled AT %ID."VF-LCR1".LASER_CONTROL_SYSTEM_POWERED_ON_I2015;
	::VFLCR_Ope0:IO.raw.iFPGARevision AT %ID."VF-LCR1".FPGA_REVISION_I2001;
	::VFLCR_Ope0:IO.ai.DMAStatus[8] AT %ID."VF-LCR1".Entry_I201A_S09;
	::VFLCR_Ope0:IO.ai.DMAStatus[7] AT %ID."VF-LCR1".Entry_I201A_S08;
	::VFLCR_Ope0:IO.ai.DMAStatus[6] AT %ID."VF-LCR1".Entry_I201A_S07;
	::VFLCR_Ope0:IO.ai.DMAStatus[5] AT %ID."VF-LCR1".Entry_I201A_S06;
	::VFLCR_Ope0:IO.ai.DMAStatus[4] AT %ID."VF-LCR1".Entry_I201A_S05;
	::VFLCR_Ope0:IO.ai.DMAStatus[3] AT %ID."VF-LCR1".Entry_I201A_S04;
	::VFLCR_Ope0:IO.ai.DMAStatus[13] AT %ID."VF-LCR1".Entry_I201A_S0E;
	::VFLCR_Ope0:IO.ai.DMAStatus[2] AT %ID."VF-LCR1".Entry_I201A_S03;
	::VFLCR_Ope0:IO.ai.DMAStatus[19] AT %ID."VF-LCR1".Entry_I201A_S14;
	::VFLCR_Ope0:IO.ai.DMAStatus[1] AT %ID."VF-LCR1".Entry_I201A_S02;
	::VFLCR_Ope0:IO.ai.DMAStatus[18] AT %ID."VF-LCR1".Entry_I201A_S13;
	::VFLCR_Ope0:IO.ai.DMAStatus[17] AT %ID."VF-LCR1".Entry_I201A_S12;
	::VFLCR_Ope0:IO.ai.DMAStatus[16] AT %ID."VF-LCR1".Entry_I201A_S11;
	::VFLCR_Ope0:IO.ai.DMAStatus[15] AT %ID."VF-LCR1".Entry_I201A_S10;
	::VFLCR_Ope0:IO.ai.DMAStatus[14] AT %ID."VF-LCR1".Entry_I201A_S0F;
	::VFLCR_Ope0:IO.raw.iLaserMainPowerEnabled AT %ID."VF-LCR1".LASER_MAIN_POWER_ON_I2016;
	::VFLCR_Ope0:IO.raw.iLaserReady_Error AT %ID."VF-LCR1".LASER_ERROR_READY_I2014;
	::VFLCR_Ope0:IO.ai.DMAStatus[20] AT %ID."VF-LCR1".Entry_I201A_S15;
	::VFLCR_Ope0:IO.ai.DMAStatus[12] AT %ID."VF-LCR1".Entry_I201A_S0D;
	::VFLCR_Ope0:IO.ai.DMACurrentTrajectory[7] AT %ID."VF-LCR1".Entry_I201B_S08;
	::VFLCR_Ope0:IO.ai.DMAStatus[0] AT %ID."VF-LCR1".Entry_I201A_S01;
	::VFLCR_Ope0:IO.ai.DMALastPacketPosition[8] AT %ID."VF-LCR1".Entry_I201C_S09;
	::VFLCR_Ope0:IO.ai.DMALastPacketPosition[7] AT %ID."VF-LCR1".Entry_I201C_S08;
	::VFLCR_Ope0:IO.ai.DMALastPacketPosition[6] AT %ID."VF-LCR1".Entry_I201C_S07;
	::VFLCR_Ope0:IO.ai.DMALastPacketPosition[5] AT %ID."VF-LCR1".Entry_I201C_S06;
	::VFLCR_Ope0:IO.ai.DMALastPacketPosition[4] AT %ID."VF-LCR1".Entry_I201C_S05;
	::VFLCR_Ope0:IO.ai.DMALastPacketPosition[3] AT %ID."VF-LCR1".Entry_I201C_S04;
	::VFLCR_Ope0:IO.ai.DMALastPacketPosition[2] AT %ID."VF-LCR1".Entry_I201C_S03;
	::VFLCR_Ope0:IO.ai.DMALastPacketPosition[19] AT %ID."VF-LCR1".Entry_I201C_S14;
	::VFLCR_Ope0:IO.ai.DMAStatus[9] AT %ID."VF-LCR1".Entry_I201A_S0A;
	::VFLCR_Ope0:IO.ai.DMALastPacketPosition[20] AT %ID."VF-LCR1".Entry_I201C_S15;
	::VFLCR_Ope0:IO.ai.DMALastPacketPosition[18] AT %ID."VF-LCR1".Entry_I201C_S13;
	::VFLCR_Ope0:IO.ai.DMALastPacketPosition[17] AT %ID."VF-LCR1".Entry_I201C_S12;
	::VFLCR_Ope0:IO.ai.DMALastPacketPosition[16] AT %ID."VF-LCR1".Entry_I201C_S11;
	::VFLCR_Ope0:IO.ai.DMALastPacketPosition[15] AT %ID."VF-LCR1".Entry_I201C_S10;
	::VFLCR_Ope0:IO.ai.DMALastPacketPosition[14] AT %ID."VF-LCR1".Entry_I201C_S0F;
	::VFLCR_Ope0:IO.ai.DMALastPacketPosition[13] AT %ID."VF-LCR1".Entry_I201C_S0E;
	::VFLCR_Ope0:IO.ai.DMALastPacketPosition[12] AT %ID."VF-LCR1".Entry_I201C_S0D;
	::VFLCR_Ope0:IO.ai.DMALastPacketPosition[11] AT %ID."VF-LCR1".Entry_I201C_S0C;
	::VFLCR_Ope0:IO.ai.DMAStatus[10] AT %ID."VF-LCR1".Entry_I201A_S0B;
	::VFLCR_Ope0:IO.ai.DMALastPacketPosition[1] AT %ID."VF-LCR1".Entry_I201C_S02;
	::VFLCR_Ope0:IO.ai.DMAStatus[11] AT %ID."VF-LCR1".Entry_I201A_S0C;
	::VFLCR_Ope0:IO.ai.DMALastPacketPosition[10] AT %ID."VF-LCR1".Entry_I201C_S0B;
	::VFLCR_Ope0:IO.ai.DMALastPacketPosition[0] AT %ID."VF-LCR1".Entry_I201C_S01;
	::VFLCR_Ope0:IO.ai.DMACurrentTrajectory[6] AT %ID."VF-LCR1".Entry_I201B_S07;
	::VFLCR_Ope0:IO.ai.DMACurrentTrajectory[5] AT %ID."VF-LCR1".Entry_I201B_S06;
	::VFLCR_Ope0:IO.ai.DMACurrentTrajectory[4] AT %ID."VF-LCR1".Entry_I201B_S05;
	::VFLCR_Ope0:IO.ai.DMACurrentTrajectory[3] AT %ID."VF-LCR1".Entry_I201B_S04;
	::VFLCR_Ope0:IO.ai.DMACurrentTrajectory[2] AT %ID."VF-LCR1".Entry_I201B_S03;
	::VFLCR_Ope0:IO.ai.DMACurrentTrajectory[20] AT %ID."VF-LCR1".Entry_I201B_S15;
	::VFLCR_Ope0:IO.ai.DMACurrentTrajectory[19] AT %ID."VF-LCR1".Entry_I201B_S14;
	::VFLCR_Ope0:IO.ai.DMACurrentTrajectory[1] AT %ID."VF-LCR1".Entry_I201B_S02;
	::VFLCR_Ope0:IO.ai.DMACurrentTrajectory[18] AT %ID."VF-LCR1".Entry_I201B_S13;
	::VFLCR_Ope0:IO.ai.DMALastPacketPosition[9] AT %ID."VF-LCR1".Entry_I201C_S0A;
	::VFLCR_Ope0:IO.ai.DMACurrentTrajectory[17] AT %ID."VF-LCR1".Entry_I201B_S12;
	::VFLCR_Ope0:IO.ai.DMACurrentTrajectory[15] AT %ID."VF-LCR1".Entry_I201B_S10;
	::VFLCR_Ope0:IO.ai.DMACurrentTrajectory[14] AT %ID."VF-LCR1".Entry_I201B_S0F;
	::VFLCR_Ope0:IO.ai.DMACurrentTrajectory[13] AT %ID."VF-LCR1".Entry_I201B_S0E;
	::VFLCR_Ope0:IO.ai.DMACurrentTrajectory[12] AT %ID."VF-LCR1".Entry_I201B_S0D;
	::VFLCR_Ope0:IO.ai.DMACurrentTrajectory[11] AT %ID."VF-LCR1".Entry_I201B_S0C;
	::VFLCR_Ope0:IO.ai.DMACurrentTrajectory[10] AT %ID."VF-LCR1".Entry_I201B_S0B;
	::VFLCR_Ope0:IO.ai.DMACurrentTrajectory[9] AT %ID."VF-LCR1".Entry_I201B_S0A;
	::VFLCR_Ope0:IO.ai.DMACurrentTrajectory[8] AT %ID."VF-LCR1".Entry_I201B_S09;
	::VFLCR_Ope0:IO.ai.DMACurrentTrajectory[16] AT %ID."VF-LCR1".Entry_I201B_S11;
	::VFLCR_Ope0:IO.raw.oIndirectRegisterRequestAddress AT %QD."VF-LCR1".REQUEST_ADDRESS_I201FOut;
	::VFLCR_Ope0:IO.raw.oIndirectRegisterRequestData AT %QD."VF-LCR1".REQUEST_DATA_I2020Out;
	::VFLCR_Ope0:IO.raw.iIndirectRegisterResponseAddress AT %ID."VF-LCR1".RESPONSE_ADDRESS_I2021;
	::VFLCR_Ope0:IO.raw.iIndirectRegisterResponseData AT %ID."VF-LCR1".RESPONSE_DATA_I2022;
	::VFLCR_Ope1:IO.raw.oIndirectRegisterRequestAddress AT %QD."VF-LCR2".REQUEST_ADDRESS_I201FOut;
	::VFLCR_Ope1:IO.raw.oIndirectRegisterRequestData AT %QD."VF-LCR2".REQUEST_DATA_I2020Out;
	::VFLCR_Ope1:IO.raw.iIndirectRegisterResponseAddress AT %ID."VF-LCR2".RESPONSE_ADDRESS_I2021;
	::VFLCR_Ope1:IO.raw.iIndirectRegisterResponseData AT %ID."VF-LCR2".RESPONSE_DATA_I2022;
	::VFLCR_Ope2:IO.raw.oIndirectRegisterRequestAddress AT %QD."VF-LCR3".REQUEST_ADDRESS_I201FOut;
	::VFLCR_Ope2:IO.raw.oIndirectRegisterRequestData AT %QD."VF-LCR3".REQUEST_DATA_I2020Out;
	::VFLCR_Ope2:IO.raw.iIndirectRegisterResponseAddress AT %ID."VF-LCR3".RESPONSE_ADDRESS_I2021;
	::VFLCR_Ope2:IO.raw.iIndirectRegisterResponseData AT %ID."VF-LCR3".RESPONSE_DATA_I2022;
	::VFLCR_Ope3:IO.raw.oIndirectRegisterRequestAddress AT %QD."VF-LCR4".REQUEST_ADDRESS_I201FOut;
	::VFLCR_Ope3:IO.raw.oIndirectRegisterRequestData AT %QD."VF-LCR4".REQUEST_DATA_I2020Out;
	::VFLCR_Ope3:IO.raw.iIndirectRegisterResponseAddress AT %ID."VF-LCR4".RESPONSE_ADDRESS_I2021;
	::VFLCR_Ope3:IO.raw.iIndirectRegisterResponseData AT %ID."VF-LCR4".RESPONSE_DATA_I2022;
END_VAR
```

- Safety project (password-protected, skipped)

## Configuration ControlPLC_DataDistribution

CPU 5PC900.TS17-02, AutomationRuntime D4.92, Build 6.3.0, Safety 0.0, Vc 

### Task classes (Cpu.sw)
```
Cyclic#1 (cycle 2000 us, tolerance 0 us):
  FirstInitP <- Infrastructure.FirstInitProg.prg
  VFLCR_HMI <- (binary)
Cyclic#2 (cycle 4000 us, tolerance 0 us):
  VFLCR_Ope0 <- ProcessControl.VFLCR.VFLCR_Operation.prg  // VF-LCR0 Operations
  VFLCR_Ope1 <- ProcessControl.VFLCR.VFLCR_Operation.prg  // VF-LCR1 Operations
  VFLCR_Ope2 <- ProcessControl.VFLCR.VFLCR_Operation.prg  // VF-LCR2 Operations
  VFLCR_Ope3 <- ProcessControl.VFLCR.VFLCR_Operation.prg  // VF-LCR3 Operations
  AlarmWrap <- Infrastructure.Alarms.AlarmWrap.prg
Cyclic#4 (cycle 12000 us, tolerance 12000 us):
  atnDriver <- Infrastructure.atnDriver.prg
  DataDis <- Automation.DataDistributionSFC.prg
  SFCControl <- Automation.SFCControl.prg
  VFLCR_Syst <- ProcessControl.VFLCR.VFLCR_System.prg  // VF-LCR System Control
  RM_BuildIn <- DataManagement.PrintJobManagement.RM_BuildInfo.prg
  RM_PrintPr <- DataManagement.PrintJobManagement.RM_PrintProcessConfig.prg
  PrintJobMa <- DataManagement.PrintJobManagement.PrintJobManagement.prg
  BuildDistr <- DataManagement.PrintJobManagement.BuildDistributor.prg
Cyclic#8 (cycle 4000 us, tolerance 32000000 us):
  RevInfo <- Infrastructure.RevInfo.RevInfo.prg
DataObjects: McAcpSys
NcDataObjects: McDriveLog
Binaries: mvLoader, TCData, FWRules, mcacpdrv, udbdef, mCoWebSc, McProfGen, TCLang, arcoal, arflatprv, arsvcreg, Role, arconfig, User, asfw, ashwd, ashwac, sysconf, iomap, MachineAH, MachineAC, MachineCG, Settings, TC, Recipies, Settings_1, UserMgmt, UserLogin, McAcpSim, McMechSys, GantryMech, RectrCfg, Hierarchy, GantryGrp, GantryCfg, CncFeature, VAx, Config, LiftCfg, ShuttleCfg, AxFeatures, asiol2, asiol1, Config_1, AirlockCfg, HopperCfg, PermMemAC, RecoaterAC, CNCAC, InitCG, PermMemCG, CNCCG, RecoaterCG, InitAC, AxBasicCG, AxBasicAC, LaserCG, LaserAC, CoolingCG, GearLiftAC, CoolingAC, VisionAC, VisionCG, FilterCG, FilterAC, PumpsAC, PumpsCG, LiftZAC, RecoatXAC, GantryXAC, GasAC, LiftCG, SafetyAC, SafetyCG, LiftAC, GasCG, GearLiftCG, GearingCG, DriversCG, DriversAC, SubsCG, SubsAC, ServoMgrCG, ServoMgrAC, gAxis
Libraries: errorAPI, McBase, SfDomain, MpBase, CoTrace, AsZip, FileIO, runtime, fiowrap, hmitools, logthat, ringbuflib, piper, DataBuffer, AsGuard, AsIODiag, sys_lib, AsBrStr, standard, AsArLog, ArEventLog, AsHttp, AsBrWStr, AsTCP, MpAxis, McAxis, MpAlarmX, stringext, bodyguard, tcpcomm, astime, McAcpAx, messagebox, MpCnc, McAxGroup, McPathGen, McProgInt, omjson, VFAlarms, MpCom, AsXml, McPureVAx, ToolBox, Finder, VF_COMMON, LoopCont, MTData, MTTypes, LoopConR, AsBrMath, MpRecipe, brsystem, VFValve, axislib, hammers, MTLookUp, AsIoTime, AsARCfg, UnitTest, UtMgr, UtWs, MpWebXs, AsArSdm, atn, MTBasics, VF_PARSER, IotMqtt, AsIecCon, ArCert, AsHW, AsETH, MpUserX, csvfilelib, persist, vartools, MpSfDomMgr, SfDomDrv, SfDomVis, asepl, powerlnk, aruser, dataobj, asusb, operator, arssl, asio, asmem, asarprof
```

### Hardware
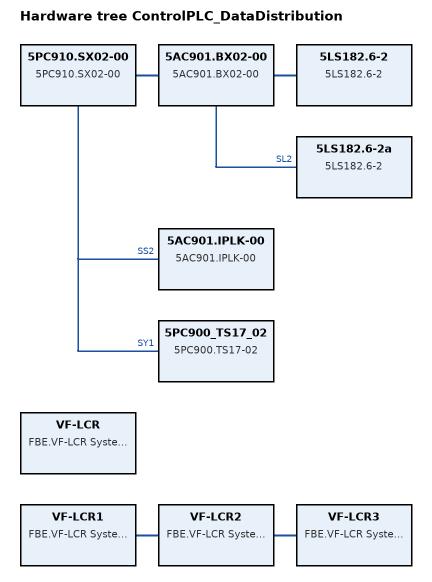
```
5AC901.BX02-00 : 5AC901.BX02-00 v1.0.1.0  [SY -> 5PC910.SX02-00.SY3]
5AC901.IPLK-00 : 5AC901.IPLK-00 v1.8.1.0  [SS -> 5PC910.SX02-00.SS2]
  Connector IF1:
    EplNatSubnet = 192.168.102.0
5LS182.6-2 : 5LS182.6-2 v1.9.0.0  [SL -> 5AC901.BX02-00.SL1]
5LS182.6-2a : 5LS182.6-2 v1.9.0.0  [SL -> 5AC901.BX02-00.SL2]
  Connector IF1:
    EplNatSubnet = 192.168.103.0
5PC900_TS17_02 : 5PC900.TS17-02 v2.1.0.0  [SY -> 5PC910.SX02-00.SY1]
  ConfigurationID = DataDistribution
  UserPartitionSize = 5000
  UserRamDevice = PCI.1.LS182.SRAM
  UserRamSize = 910000
  RemMemDevice = PCI.1.LS182.SRAM
  RemMemSize = 116736
  PermanentPvSize = 30000
  RemanentGlobalPvSize = 85000
  VolatileGlobalPvSize = 1100000
  ClearNvMemoryAfterShutdownFlushError = 0
  CyclicFlushRemMemSelector = 1
  SystemLoggerSize = 512000
  FieldbusLoggerSize = 102400
  SafetyLoggerSize = 512000
  ConnectivityLoggerSize = 102400
  AccessAndSecurityLoggerSize = 102400
  TextSystemLoggerSize = 51200
  UnitSystemLoggerSize = 51200
  FirewallLoggerSize = 51200
  UserLoggerSize = 512000
  RebootReset = 1
  IdleTaskClass = 3
  TaskClassIdleTime = 2000
  Cyclic1Duration = 2000
  Cyclic1Tolerance = 0
  Cyclic1Output = 1
  Cyclic2Duration = 4000
  Cyclic2Tolerance = 0
  Cyclic3Duration = 6000
  Cyclic3Tolerance = 0
  Cyclic4Duration = 12000
  Cyclic4Tolerance = 12000
  Cyclic5Duration = 52000
  Cyclic5Tolerance = 52000
  Cyclic6Duration = 102000
  Cyclic6Tolerance = 102000
  Cyclic7Duration = 410000
  Cyclic7Tolerance = 410000
  Cyclic8Duration = 4000
  Cyclic8Tolerance = 32000000
  FileDevice1
  FileDeviceName1 = USER
  FileDevicePath1 = USER_PATH
  TimeZone = 65
  ActivateDaylightSavingTime = 1
  ActivateSntp = 1
  SntpcServAddr1 = 192.168.200.30
  FtpUser1
  FtpUsername1 = admin
  FtpUserPassword1 = exkK5AJZIoUR27ZAGAewwmn6IiVY4aYFmsGoBfzbjRw=  // VFftp
  FtpUserSalt1 = qubFqNjb
  FTPAccessRight1 = 0
  FTPdevice1 = ALL
  ActivateOpcUa = 1
  OpcUa_ConversationSecurityPolicy_EnableBasic128Rsa15 = 0
  OpcUa_AuthenticationSecurityPolicy_EnableNone = 1
  OpcUa_Security_AdminRole = Administrators
  OpcUaLimitsMaxPublish = 50
  OpcUa_SamplingTimer_Default = 5
  OpcUa_SamplingTimer6_Interval = 1000
  OpcUa_SamplingTimer7_Interval = 5000
  OpcUa_SamplingTimer8_Interval = 10000
  OpcUaInformationModels_PV_Version = 2
5PC910.SX02-00 : 5PC910.SX02-00 v2.1.2.0
  Connector IF1:
    AssignedOperatingSystem = ARemb
  Connector IF3:
    AssignedOperatingSystem = ARemb
    ActivateDevice = 1
    Mode = Manual
    InternetAddress = 192.168.200.50
    SubnetMask = 255.255.255.0
  Connector IF4:
    AssignedOperatingSystem = ARemb
    ActivateDevice = 1
  Connector IF5:
    AssignedOperatingSystem = ARemb
  Connector IF6:
    AssignedOperatingSystem = ARemb
  Connector IF7:
    AssignedOperatingSystem = ARemb
  Connector IF8:
    AssignedOperatingSystem = ARemb
  Connector IF9:
    AssignedOperatingSystem = ARemb
VF-LCR : FBE.VF-LCR System (version 04) v04 (OrderNumber=VF-LCR)  [PLK1 -> VF-LCR3.PLK2 (NodeNumber=51) [Cable Type=PowerlinkCable, Length=10, Version=1.0.0.3]; PLK2 -> 5LS182.6-2.IF1 (NodeNumber=51) [Cable Type=PowerlinkCable, Length=10, Version=1.0.0.3]]
  Supervision = off
  ResponseTimeout = 50
VF-LCR1 : FBE.VF-LCR System (version 04) v04 (OrderNumber=VF-LCR)  [PLK2 -> VF-LCR2.PLK1 (NodeNumber=52) [Cable Type=PowerlinkCable, Length=10, Version=1.0.0.3]]
  Supervision = off
  ResponseTimeout = 50
VF-LCR2 : FBE.VF-LCR System (version 04) v04 (OrderNumber=VF-LCR)  [PLK1 -> VF-LCR1.PLK2 (NodeNumber=53) [Cable Type=PowerlinkCable, Length=10, Version=1.0.0.3]; PLK2 -> VF-LCR3.PLK1 (NodeNumber=53) [Cable Type=PowerlinkCable, Length=10, Version=1.0.0.3]]
  Supervision = off
  ResponseTimeout = 50
VF-LCR3 : FBE.VF-LCR System (version 04) v04 (OrderNumber=VF-LCR)  [PLK1 -> VF-LCR2.PLK2 (NodeNumber=54) [Cable Type=PowerlinkCable, Length=10, Version=1.0.0.3]; PLK2 -> VF-LCR.PLK1 (NodeNumber=54) [Cable Type=PowerlinkCable, Length=10, Version=1.0.0.3]]
  Supervision = off
  ResponseTimeout = 50
```

### IoMap.iom - 5PC900_TS17_02/IoMap.iom
```iecst
VAR_CONFIG
	::VFLCR_Ope0:IO.raw.oSystemControl AT %QD."VF-LCR".SYSTEM_CONTROL_I2004Out;
	::VFLCR_Ope0:IO.ao.SelectedPrintNumber AT %QD."VF-LCR".SELECTED_PRINT_NUMBER_I200BOut;
	::VFLCR_Ope0:IO.ao.SelectedLayerNumber AT %QD."VF-LCR".SELECTED_LAYER_NUMBER_I200COut;
	::VFLCR_Ope0:IO.ao.SelectedBuildLayout AT %QD."VF-LCR".SELECTED_BUILD_LAYOUT_I200AOut;
	::VFLCR_Ope0:IO.ao.PLCHeartbeat AT %QD."VF-LCR".PLC_HEARTBEAT_I2003Out;
	::VFLCR_Ope0:IO.raw.oOperationControl AT %QD."VF-LCR".OPERATION_CONTROL_I2005Out;
	::VFLCR_Ope0:IO.raw.oManualLaserOperation AT %QD."VF-LCR".MANUAL_LASER_OPERATION_I200EOut;
	::VFLCR_Ope0:IO.raw.oManualLaserCurrentSetpoint AT %QD."VF-LCR".MANUAL_LASER_CURRENT_SETPOINT_I200FOut;
	::VFLCR_Ope0:IO.raw.oLaserEnable AT %QD."VF-LCR".LASER_ENABLE_I2008Out;
	::VFLCR_Ope0:IO.raw.oEnableLaserMainPower AT %QD."VF-LCR".LASER_REMOTE_START_I2010Out;
	::VFLCR_Ope0:IO.raw.oEnableLaserEmission AT %QD."VF-LCR".LASER_EMISSION_CONTROL_I2012Out;
	::VFLCR_Ope0:IO.raw.oEnableGuideLaser AT %QD."VF-LCR".GUIDE_LASER_CONTROL_I2011Out;
	::VFLCR_Ope0:IO.raw.oResetLaserErrors AT %QD."VF-LCR".LASER_RESET_I2013Out;
	::VFLCR_Ope0:IO.di.PoweLinkModuleOK AT %IX."VF-LCR".ModuleOk;
	::VFLCR_Ope0:IO.raw.iLaserFatalError AT %ID."VF-LCR".SYSTEM_ERROR_I2018;
	::VFLCR_Ope0:IO.raw.iSystemStatus AT %ID."VF-LCR".SYSTEM_STATUS_I2006;
	::VFLCR_Ope0:IO.ai.SystemHeartbeat AT %ID."VF-LCR".SYSTEM_HEARTBEAT_I2002;
	::VFLCR_Ope0:IO.raw.iSoftwareRevision AT %ID."VF-LCR".SOFTWARE_REVISION_I201D;
	::VFLCR_Ope0:IO.raw.iOperationStatus AT %ID."VF-LCR".OPERATION_STATUS_I2007;
	::VFLCR_Ope0:IO.raw.iManualModeLaserPower AT %ID."VF-LCR".LASER_POWER_MONITOR_I2019;
	::VFLCR_Ope0:IO.ai.LUTFiles_CalibrationID AT %ID."VF-LCR".LUT_LOAD_STATUS_I2009;
	::VFLCR_Ope0:IO.raw.iLaserWatchdogError AT %ID."VF-LCR".LASER_WATCHDOG_ERROR_I201E;
	::VFLCR_Ope0:IO.raw.iLaserEmissionEnabled AT %ID."VF-LCR".LASER_EMISSION_ON_I2017;
	::VFLCR_Ope0:IO.raw.iLaserControlPowerEnabled AT %ID."VF-LCR".LASER_CONTROL_SYSTEM_POWERED_ON_I2015;
	::VFLCR_Ope0:IO.raw.iFPGARevision AT %ID."VF-LCR".FPGA_REVISION_I2001;
	::VFLCR_Ope0:IO.raw.iLaserMainPowerEnabled AT %ID."VF-LCR".LASER_MAIN_POWER_ON_I2016;
	::VFLCR_Ope0:IO.raw.iLaserReady_Error AT %ID."VF-LCR".LASER_ERROR_READY_I2014;
	::VFLCR_Ope1:IO.raw.oSystemControl AT %QD."VF-LCR1".SYSTEM_CONTROL_I2004Out;
	::VFLCR_Ope1:IO.ao.SelectedPrintNumber AT %QD."VF-LCR1".SELECTED_PRINT_NUMBER_I200BOut;
	::VFLCR_Ope1:IO.ao.SelectedLayerNumber AT %QD."VF-LCR1".SELECTED_LAYER_NUMBER_I200COut;
	::VFLCR_Ope1:IO.ao.SelectedBuildLayout AT %QD."VF-LCR1".SELECTED_BUILD_LAYOUT_I200AOut;
	::VFLCR_Ope1:IO.ao.PLCHeartbeat AT %QD."VF-LCR1".PLC_HEARTBEAT_I2003Out;
	::VFLCR_Ope1:IO.raw.oOperationControl AT %QD."VF-LCR1".OPERATION_CONTROL_I2005Out;
	::VFLCR_Ope1:IO.raw.oManualLaserOperation AT %QD."VF-LCR1".MANUAL_LASER_OPERATION_I200EOut;
	::VFLCR_Ope1:IO.raw.oManualLaserCurrentSetpoint AT %QD."VF-LCR1".MANUAL_LASER_CURRENT_SETPOINT_I200FOut;
	::VFLCR_Ope1:IO.raw.oLaserEnable AT %QD."VF-LCR1".LASER_ENABLE_I2008Out;
	::VFLCR_Ope1:IO.raw.oEnableLaserMainPower AT %QD."VF-LCR1".LASER_REMOTE_START_I2010Out;
	::VFLCR_Ope1:IO.raw.oEnableLaserEmission AT %QD."VF-LCR1".LASER_EMISSION_CONTROL_I2012Out;
	::VFLCR_Ope1:IO.raw.oEnableGuideLaser AT %QD."VF-LCR1".GUIDE_LASER_CONTROL_I2011Out;
	::VFLCR_Ope1:IO.raw.oResetLaserErrors AT %QD."VF-LCR1".LASER_RESET_I2013Out;
	::VFLCR_Ope1:IO.di.PoweLinkModuleOK AT %IX."VF-LCR1".ModuleOk;
	::VFLCR_Ope1:IO.raw.iLaserFatalError AT %ID."VF-LCR1".SYSTEM_ERROR_I2018;
	::VFLCR_Ope1:IO.raw.iSystemStatus AT %ID."VF-LCR1".SYSTEM_STATUS_I2006;
	::VFLCR_Ope1:IO.ai.SystemHeartbeat AT %ID."VF-LCR1".SYSTEM_HEARTBEAT_I2002;
	::VFLCR_Ope1:IO.raw.iSoftwareRevision AT %ID."VF-LCR1".SOFTWARE_REVISION_I201D;
	::VFLCR_Ope1:IO.raw.iOperationStatus AT %ID."VF-LCR1".OPERATION_STATUS_I2007;
	::VFLCR_Ope1:IO.raw.iManualModeLaserPower AT %ID."VF-LCR1".LASER_POWER_MONITOR_I2019;
	::VFLCR_Ope1:IO.ai.LUTFiles_CalibrationID AT %ID."VF-LCR1".LUT_LOAD_STATUS_I2009;
	::VFLCR_Ope1:IO.raw.iLaserWatchdogError AT %ID."VF-LCR1".LASER_WATCHDOG_ERROR_I201E;
	::VFLCR_Ope1:IO.raw.iLaserEmissionEnabled AT %ID."VF-LCR1".LASER_EMISSION_ON_I2017;
	::VFLCR_Ope1:IO.raw.iLaserControlPowerEnabled AT %ID."VF-LCR1".LASER_CONTROL_SYSTEM_POWERED_ON_I2015;
	::VFLCR_Ope1:IO.raw.iFPGARevision AT %ID."VF-LCR1".FPGA_REVISION_I2001;
	::VFLCR_Ope1:IO.raw.iLaserMainPowerEnabled AT %ID."VF-LCR1".LASER_MAIN_POWER_ON_I2016;
	::VFLCR_Ope1:IO.raw.iLaserReady_Error AT %ID."VF-LCR1".LASER_ERROR_READY_I2014;
	::VFLCR_Ope2:IO.raw.oSystemControl AT %QD."VF-LCR2".SYSTEM_CONTROL_I2004Out;
	::VFLCR_Ope2:IO.ao.SelectedPrintNumber AT %QD."VF-LCR2".SELECTED_PRINT_NUMBER_I200BOut;
	::VFLCR_Ope2:IO.ao.SelectedLayerNumber AT %QD."VF-LCR2".SELECTED_LAYER_NUMBER_I200COut;
	::VFLCR_Ope2:IO.ao.SelectedBuildLayout AT %QD."VF-LCR2".SELECTED_BUILD_LAYOUT_I200AOut;
	::VFLCR_Ope2:IO.ao.PLCHeartbeat AT %QD."VF-LCR2".PLC_HEARTBEAT_I2003Out;
	::VFLCR_Ope2:IO.raw.oOperationControl AT %QD."VF-LCR2".OPERATION_CONTROL_I2005Out;
	::VFLCR_Ope2:IO.raw.oManualLaserOperation AT %QD."VF-LCR2".MANUAL_LASER_OPERATION_I200EOut;
	::VFLCR_Ope2:IO.raw.oManualLaserCurrentSetpoint AT %QD."VF-LCR2".MANUAL_LASER_CURRENT_SETPOINT_I200FOut;
	::VFLCR_Ope2:IO.raw.oLaserEnable AT %QD."VF-LCR2".LASER_ENABLE_I2008Out;
	::VFLCR_Ope2:IO.raw.oEnableLaserMainPower AT %QD."VF-LCR2".LASER_REMOTE_START_I2010Out;
	::VFLCR_Ope2:IO.raw.oEnableLaserEmission AT %QD."VF-LCR2".LASER_EMISSION_CONTROL_I2012Out;
	::VFLCR_Ope2:IO.raw.oEnableGuideLaser AT %QD."VF-LCR2".GUIDE_LASER_CONTROL_I2011Out;
	::VFLCR_Ope2:IO.raw.oResetLaserErrors AT %QD."VF-LCR2".LASER_RESET_I2013Out;
	::VFLCR_Ope2:IO.di.PoweLinkModuleOK AT %IX."VF-LCR2".ModuleOk;
	::VFLCR_Ope2:IO.raw.iLaserFatalError AT %ID."VF-LCR2".SYSTEM_ERROR_I2018;
	::VFLCR_Ope2:IO.raw.iSystemStatus AT %ID."VF-LCR2".SYSTEM_STATUS_I2006;
	::VFLCR_Ope2:IO.ai.SystemHeartbeat AT %ID."VF-LCR2".SYSTEM_HEARTBEAT_I2002;
	::VFLCR_Ope2:IO.raw.iSoftwareRevision AT %ID."VF-LCR2".SOFTWARE_REVISION_I201D;
	::VFLCR_Ope2:IO.raw.iOperationStatus AT %ID."VF-LCR2".OPERATION_STATUS_I2007;
	::VFLCR_Ope2:IO.raw.iManualModeLaserPower AT %ID."VF-LCR2".LASER_POWER_MONITOR_I2019;
	::VFLCR_Ope2:IO.ai.LUTFiles_CalibrationID AT %ID."VF-LCR2".LUT_LOAD_STATUS_I2009;
	::VFLCR_Ope2:IO.raw.iLaserWatchdogError AT %ID."VF-LCR2".LASER_WATCHDOG_ERROR_I201E;
	::VFLCR_Ope2:IO.raw.iLaserEmissionEnabled AT %ID."VF-LCR2".LASER_EMISSION_ON_I2017;
	::VFLCR_Ope2:IO.raw.iLaserControlPowerEnabled AT %ID."VF-LCR2".LASER_CONTROL_SYSTEM_POWERED_ON_I2015;
	::VFLCR_Ope2:IO.raw.iFPGARevision AT %ID."VF-LCR2".FPGA_REVISION_I2001;
	::VFLCR_Ope2:IO.raw.iLaserMainPowerEnabled AT %ID."VF-LCR2".LASER_MAIN_POWER_ON_I2016;
	::VFLCR_Ope2:IO.raw.iLaserReady_Error AT %ID."VF-LCR2".LASER_ERROR_READY_I2014;
	::VFLCR_Ope3:IO.raw.oSystemControl AT %QD."VF-LCR3".SYSTEM_CONTROL_I2004Out;
	::VFLCR_Ope3:IO.ao.SelectedPrintNumber AT %QD."VF-LCR3".SELECTED_PRINT_NUMBER_I200BOut;
	::VFLCR_Ope3:IO.ao.SelectedLayerNumber AT %QD."VF-LCR3".SELECTED_LAYER_NUMBER_I200COut;
	::VFLCR_Ope3:IO.ao.SelectedBuildLayout AT %QD."VF-LCR3".SELECTED_BUILD_LAYOUT_I200AOut;
	::VFLCR_Ope3:IO.ao.PLCHeartbeat AT %QD."VF-LCR3".PLC_HEARTBEAT_I2003Out;
	::VFLCR_Ope3:IO.raw.oOperationControl AT %QD."VF-LCR3".OPERATION_CONTROL_I2005Out;
	::VFLCR_Ope3:IO.raw.oManualLaserOperation AT %QD."VF-LCR3".MANUAL_LASER_OPERATION_I200EOut;
	::VFLCR_Ope3:IO.raw.oManualLaserCurrentSetpoint AT %QD."VF-LCR3".MANUAL_LASER_CURRENT_SETPOINT_I200FOut;
	::VFLCR_Ope3:IO.raw.oLaserEnable AT %QD."VF-LCR3".LASER_ENABLE_I2008Out;
	::VFLCR_Ope3:IO.raw.oEnableLaserMainPower AT %QD."VF-LCR3".LASER_REMOTE_START_I2010Out;
	::VFLCR_Ope3:IO.raw.oEnableLaserEmission AT %QD."VF-LCR3".LASER_EMISSION_CONTROL_I2012Out;
	::VFLCR_Ope3:IO.raw.oEnableGuideLaser AT %QD."VF-LCR3".GUIDE_LASER_CONTROL_I2011Out;
	::VFLCR_Ope3:IO.raw.oResetLaserErrors AT %QD."VF-LCR3".LASER_RESET_I2013Out;
	::VFLCR_Ope3:IO.di.PoweLinkModuleOK AT %IX."VF-LCR3".ModuleOk;
	::VFLCR_Ope3:IO.raw.iLaserFatalError AT %ID."VF-LCR3".SYSTEM_ERROR_I2018;
	::VFLCR_Ope3:IO.raw.iSystemStatus AT %ID."VF-LCR3".SYSTEM_STATUS_I2006;
	::VFLCR_Ope3:IO.ai.SystemHeartbeat AT %ID."VF-LCR3".SYSTEM_HEARTBEAT_I2002;
	::VFLCR_Ope3:IO.raw.iSoftwareRevision AT %ID."VF-LCR3".SOFTWARE_REVISION_I201D;
	::VFLCR_Ope3:IO.raw.iOperationStatus AT %ID."VF-LCR3".OPERATION_STATUS_I2007;
	::VFLCR_Ope3:IO.raw.iManualModeLaserPower AT %ID."VF-LCR3".LASER_POWER_MONITOR_I2019;
	::VFLCR_Ope3:IO.ai.LUTFiles_CalibrationID AT %ID."VF-LCR3".LUT_LOAD_STATUS_I2009;
	::VFLCR_Ope3:IO.raw.iLaserWatchdogError AT %ID."VF-LCR3".LASER_WATCHDOG_ERROR_I201E;
	::VFLCR_Ope3:IO.raw.iLaserEmissionEnabled AT %ID."VF-LCR3".LASER_EMISSION_ON_I2017;
	::VFLCR_Ope3:IO.raw.iLaserControlPowerEnabled AT %ID."VF-LCR3".LASER_CONTROL_SYSTEM_POWERED_ON_I2015;
	::VFLCR_Ope3:IO.raw.iFPGARevision AT %ID."VF-LCR3".FPGA_REVISION_I2001;
	::VFLCR_Ope3:IO.raw.iLaserMainPowerEnabled AT %ID."VF-LCR3".LASER_MAIN_POWER_ON_I2016;
	::VFLCR_Ope3:IO.raw.iLaserReady_Error AT %ID."VF-LCR3".LASER_ERROR_READY_I2014;
END_VAR
```

### MachineAH.mpalarmxhistory - 5PC900_TS17_02/mappServices/MachineAH.mpalarmxhistory
```
Element gAlarmXHistory_Machine (Type=mpalarmxhistory)
```

### Recipies.mprecipexml - 5PC900_TS17_02/mappServices/Recipies.mprecipexml
```
Element gBuildInfoRecipe (Type=mprecipexml)
  Alarms = MpAlarmX
    mapp.AlarmX.Core.Configuration:
      [0]:
        Code = 1300
        Severity = 4
        AdditionalInformation1 = Build Info
        AdditionalInformation2 = Recipe
      [1]:
        Code = 1301
        Severity = 4
        AdditionalInformation1 = Build Info
        AdditionalInformation2 = Recipe
      [2]:
        Code = 1302
        Severity = 4
        AdditionalInformation1 = Build Info
        AdditionalInformation2 = Recipe
      [3]:
        Code = 1303
        Severity = 4
        AdditionalInformation1 = Build Info
        AdditionalInformation2 = Recipe
Element gCustomScanRecipe (Type=mprecipexml)
  Alarms = MpAlarmX
Element gPrintProcessConfigRecipe (Type=mprecipexml)
  Alarms = MpAlarmX
```

### UserMgmt.mpuserx - 5PC900_TS17_02/mappServices/UserMgmt.mpuserx
```
Element UserMgmtX (Type=mpuserx)
  Mgr:
    PasswordLength = 1
    LoginAttempts = 10
    SignAttempts = 10
  ServerSettings:
    Server:
      AdditionalUserData:
        [0] = mail
        [1] = telephoneNumber
  Users:
    DefUser#1:
      id = Key1
    DefUser#2:
      id = Key2
    DefUser#3:
      id = Key3
    DefUser#4:
      id = Key4
    DefUser#5:
      id = Key5
    DefUser#6:
      id = Key6
    DefUser#7:
      id = Key7
    DefUser#8:
      id = Key8
    DefUser#9:
      id = Key9
    DefUser#10:
      id = Key10
    DefUser#11:
      id = Remote
    DefUser#12:
      id = Operator
    DefUser#13:
      id = Manufacturing
    DefUser#14:
      id = Mechanical Engineer
    DefUser#15:
      id = Controls Engineer
  Groups:
    DefGroup#1:
      id = AccessLevel1
      level = 1
    DefGroup#2:
      id = AccessLevel2
      level = 2
    DefGroup#3:
      id = AccessLevel3
      level = 3
    DefGroup#4:
      id = AccessLevel4
      level = 4
    DefGroup#5:
      id = AccessLevel5
      level = 5
    DefGroup#6:
      id = AccessLevel6
      level = 6
    DefGroup#7:
      id = AccessLevel7
      level = 7
    DefGroup#8:
      id = AccessLevel8
      level = 8
    DefGroup#9:
      id = AccessLevel9
      level = 9
    DefGroup#10:
      id = AccessLevel10
      admin = TRUE
    DefGroup#11:
      id = Remote
      level = 1
    DefGroup#12:
      id = Operators
      level = 2
    DefGroup#13:
      id = Manufacturing
      level = 5
    DefGroup#14:
      id = Mechanical Engineer
      level = 9
    DefGroup#15:
      id = Controls Engineer
      admin = TRUE
```

## Configuration ControlPLC_LaserCleanroom

CPU 5PC900.TS17-02, AutomationRuntime C4.92, Build 6.3.0, Safety 0.0, Vc 

### Task classes (Cpu.sw)
```
Cyclic#1 (cycle 2000 us, tolerance 0 us):
  FirstInitP <- Infrastructure.FirstInitProg.prg
  VFPTR_Syst <- ProcessControl.VFLCR.VFPTR_System.prg  // VF-PTR System Control
  VFLCR_HMI <- (binary)
Cyclic#2 (cycle 4000 us, tolerance 0 us):
  VFLCR_Alar <- ProcessControl.VFLCR.VFLCR_Alarm.prg
  VFLCR_Ope0 <- ProcessControl.VFLCR.VFLCR_Operation.prg  // VF-LCR0 Operations
  VFLCR_Ope1 <- ProcessControl.VFLCR.VFLCR_Operation.prg  // VF-LCR1 Operations
  VFLCR_Ope2 <- ProcessControl.VFLCR.VFLCR_Operation.prg  // VF-LCR2 Operations
  VFLCR_Ope3 <- ProcessControl.VFLCR.VFLCR_Operation.prg  // VF-LCR3 Operations
  AlarmWrap <- Infrastructure.Alarms.AlarmWrap.prg
Cyclic#4 (cycle 12000 us, tolerance 12000 us):
  atnDriver <- Infrastructure.atnDriver.prg
  ManualPuls <- Automation.ManualPulseLaserSFC.prg
  LaserGen3S <- Automation.LaserGen3SFC.prg
  SFCControl <- Automation.SFCControl.prg
  VFLCR_Syst <- ProcessControl.VFLCR.VFLCR_System.prg  // VF-LCR System Control
  MachineMod <- MachineControl.MachineMode.MachineMode.prg
  Gen3Python <- ProcessControl.VFLCR.Gen3PythonLaserCalibration.prg
  Safety <- MachineControl.Safety.Safety.prg
  TempSensor <- ProcessControl.OpticsBox.TempFlowSensors.prg
Cyclic#8 (cycle 4000 us, tolerance 32000000 us):
  VFLCR_Pixe <- ProcessControl.VFLCR.VFLCR_PixelMapping.prg
  RevInfo <- Infrastructure.RevInfo.RevInfo.prg
DataObjects: McAcpSys
NcDataObjects: McDriveLog
Binaries: mvLoader, TCData, FWRules, mcacpdrv, udbdef, mCoWebSc, McAcpSim, McMechSys, McProfGen, TCLang, arcoal, arflatprv, arsvcreg, Role, arconfig, User, asfw, ashwd, ashwac, sysconf, iomap, GantryMech, RectrCfg, MachineAH, MachineAC, Hierarchy, MachineCG, GantryGrp, GantryCfg, CncFeature, VAx, Config, LiftCfg, Settings, ShuttleCfg, AxFeatures, TC, Recipies, asiol2, asiol1, Settings_1, Config_1, AirlockCfg, UserMgmt, UserLogin, HopperCfg, PermMemAC, RecoaterAC, CNCAC, InitCG, PermMemCG, CNCCG, RecoaterCG, InitAC, AxBasicCG, AxBasicAC, LaserCG, LaserAC, CoolingCG, GearLiftAC, CoolingAC, VisionAC, VisionCG, FilterCG, FilterAC, PumpsAC, PumpsCG, LiftZAC, RecoatXAC, GantryXAC, GasAC, LiftCG, SafetyAC, SafetyCG, LiftAC, GasCG, GearLiftCG, GearingCG, DriversCG, DriversAC, SubsCG, SubsAC, ServoMgrCG, ServoMgrAC, gAxis
Libraries: errorAPI, McBase, SfDomain, MpBase, CoTrace, AsZip, FileIO, runtime, fiowrap, hmitools, logthat, ringbuflib, piper, DataBuffer, AsGuard, AsIODiag, sys_lib, AsBrStr, standard, AsArLog, ArEventLog, AsHttp, AsBrWStr, AsTCP, MpAxis, McAxis, MpAlarmX, stringext, bodyguard, tcpcomm, astime, McAcpAx, messagebox, MpCnc, McAxGroup, McPathGen, McProgInt, omjson, VFAlarms, MpCom, AsXml, McPureVAx, ToolBox, Finder, VF_COMMON, LoopCont, MTData, MTTypes, LoopConR, AsBrMath, MpRecipe, brsystem, VFValve, axislib, hammers, MTLookUp, AsIoTime, AsARCfg, UnitTest, UtMgr, UtWs, MpWebXs, AsArSdm, atn, MTBasics, VF_PARSER, IotMqtt, AsIecCon, ArCert, AsHW, AsETH, MpUserX, csvfilelib, persist, vartools, MpSfDomMgr, SfDomDrv, SfDomVis, asepl, powerlnk, aruser, dataobj, asusb, operator, arssl, asio, asmem, asarprof
```

### Hardware
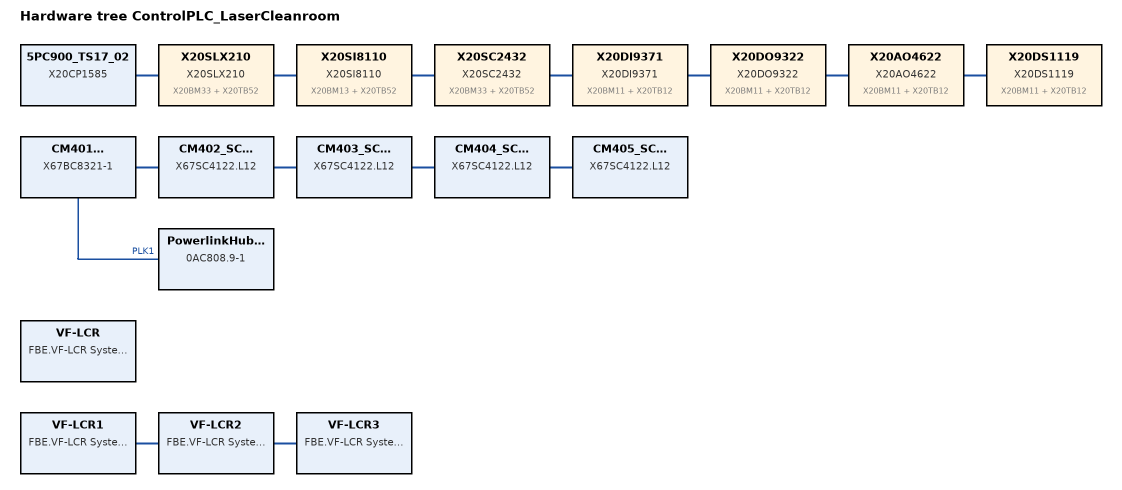
```
5PC900_TS17_02 : X20CP1585 v1.10.0.0
  Connector IF2:
    ActivateDevice = 1
    HostName = vf_main
    Mode = Manual
    InternetAddress = 192.168.200.50
    SubnetMask = 255.255.255.0
    ActivateModbus = 1
    NumSlaves = -1
    NumAllBlocks = -1
    MemSizeIn = -1
    MemSizeOut = -1
  ConfigurationID = PlatformGen3
  ConfigVersion = 3.0.0
  UserPartitionSize = 5000
  Simulation = 1
  UserRamSize = 910000
  RemMemSize = 116736
  PermanentPvSize = 30000
  RemanentGlobalPvSize = 85000
  VolatileGlobalPvSize = 1100000
  ClearNvMemoryAfterShutdownFlushError = 0
  CyclicFlushRemMemSelector = 1
  SystemLoggerSize = 512000
  FieldbusLoggerSize = 102400
  SafetyLoggerSize = 512000
  ConnectivityLoggerSize = 102400
  AccessAndSecurityLoggerSize = 102400
  TextSystemLoggerSize = 51200
  UnitSystemLoggerSize = 51200
  FirewallLoggerSize = 51200
  UserLoggerSize = 512000
  RebootReset = 1
  Connections = 5
  TimerDeviceType = EPLX2X
  TimerDevice = 5PC900_TS17_02.IF3
  IdleTaskClass = 3
  TaskClassIdleTime = 2000
  Cyclic1Duration = 2000
  Cyclic1Tolerance = 0
  Cyclic1Output = 1
  Cyclic2Duration = 4000
  Cyclic2Tolerance = 0
  Cyclic3Duration = 6000
  Cyclic3Tolerance = 0
  Cyclic4Duration = 12000
  Cyclic4Tolerance = 12000
  Cyclic5Duration = 52000
  Cyclic5Tolerance = 52000
  Cyclic6Duration = 102000
  Cyclic6Tolerance = 102000
  Cyclic7Duration = 410000
  Cyclic7Tolerance = 410000
  Cyclic8Duration = 4000
  Cyclic8Tolerance = 32000000
  FileDevice1
  FileDeviceName1 = USER
  FileDevicePath1 = USER_PATH
  TimeZone = 65
  ActivateDaylightSavingTime = 1
  ActivateSntp = 1
  SntpcServAddr1 = 192.168.200.30
  EthernetHostName = vf_main
  FtpUser1
  FtpUsername1 = admin
  FtpUserPassword1 = exkK5AJZIoUR27ZAGAewwmn6IiVY4aYFmsGoBfzbjRw=  // VFftp
  FtpUserSalt1 = qubFqNjb
  FTPAccessRight1 = 0
  FTPdevice1 = ALL
  ActivateOpcUa = 1
  OpcUaPort = 4850
  OpcUa_ConversationSecurityPolicy_EnableBasic128Rsa15 = 0
  OpcUa_AuthenticationSecurityPolicy_EnableNone = 1
  OpcUa_Security_AdminRole = Administrators
  OpcUaLimitsMaxPublish = 50
  OpcUa_SamplingTimer_Default = 5
  OpcUa_SamplingTimer6_Interval = 1000
  OpcUa_SamplingTimer7_Interval = 5000
  OpcUa_SamplingTimer8_Interval = 10000
  OpcUaInformationModels_PV_Version = 2
CM401_LaserRacks_WaterPressureOK : X67BC8321-1 v2.11.1.0  [PLK1 -> PowerlinkHub_DCEnclosure.ETH3 (NodeNumber=4) [Cable Type=PowerlinkCable, Length=10, Version=1.0.0.3]]
  Connector IF1:
    CycleTime = 800
  IOSupervision = off
CM402_SC_LaserRack1 : X67SC4122.L12 v2.2.0.0  [X2X1 -> CM401_LaserRacks_WaterPressureOK.IF1 [Cable Type=X2XCable, Length=10, Version=1.0.0.3]]
  Supervision = off
  SafeModuleID = 41
  DigitalOutput01 = viaSafeLOGIC
  DigitalOutput02 = viaSafeLOGIC
  DigitalOutput03 = viaSafeLOGIC
  DigitalOutput04 = viaSafeLOGIC
CM403_SC_LaserRack2 : X67SC4122.L12 v2.2.0.0  [X2X1 -> CM402_SC_LaserRack1.X2X2 [Cable Type=X2XCable, Length=10, Version=1.0.0.3]]
  Supervision = off
  SafeModuleID = 42
  DigitalOutput01 = viaSafeLOGIC
  DigitalOutput02 = viaSafeLOGIC
  DigitalOutput03 = viaSafeLOGIC
  DigitalOutput04 = viaSafeLOGIC
CM404_SC_LaserRack3 : X67SC4122.L12 v2.2.0.0  [X2X1 -> CM403_SC_LaserRack2.X2X2 [Cable Type=X2XCable, Length=10, Version=1.0.0.3]]
  Supervision = off
  SafeModuleID = 43
  DigitalOutput01 = viaSafeLOGIC
  DigitalOutput02 = viaSafeLOGIC
  DigitalOutput03 = viaSafeLOGIC
  DigitalOutput04 = viaSafeLOGIC
CM405_SC_LaserRack4 : X67SC4122.L12 v2.2.0.0  [X2X1 -> CM404_SC_LaserRack3.X2X2 [Cable Type=X2XCable, Length=10, Version=1.0.0.3]]
  Supervision = off
  SafeModuleID = 44
  DigitalOutput01 = viaSafeLOGIC
  DigitalOutput02 = viaSafeLOGIC
  DigitalOutput03 = viaSafeLOGIC
  DigitalOutput04 = viaSafeLOGIC
PowerlinkHub_DCEnclosure : 0AC808.9-1 v1.0.0.0  [ETH3 -> CM401_LaserRacks_WaterPressureOK.PLK1 [Cable Type=PowerlinkCable, Length=10, Version=1.0.0.3]; ETH5 -> 5PC900_TS17_02.IF3 [Cable Type=PowerlinkCable, Length=10, Version=1.0.0.3]; ETH6 -> VF-LCR.PLK2 [Cable Type=PowerlinkCable, Length=10, Version=1.0.0.3]]
VF-LCR : FBE.VF-LCR System (version 04) v04 (OrderNumber=VF-LCR)  [PLK1 -> VF-LCR3.PLK2 (NodeNumber=51) [Cable Type=PowerlinkCable, Length=10, Version=1.0.0.3]; PLK2 -> PowerlinkHub_DCEnclosure.ETH6 (NodeNumber=51) [Cable Type=PowerlinkCable, Length=10, Version=1.0.0.3]]
  Supervision = off
  ResponseTimeout = 50
VF-LCR1 : FBE.VF-LCR System (version 04) v04 (OrderNumber=VF-LCR)  [PLK2 -> VF-LCR2.PLK1 (NodeNumber=52) [Cable Type=PowerlinkCable, Length=10, Version=1.0.0.3]]
  Supervision = off
  ResponseTimeout = 50
VF-LCR2 : FBE.VF-LCR System (version 04) v04 (OrderNumber=VF-LCR)  [PLK1 -> VF-LCR1.PLK2 (NodeNumber=53) [Cable Type=PowerlinkCable, Length=10, Version=1.0.0.3]; PLK2 -> VF-LCR3.PLK1 (NodeNumber=53) [Cable Type=PowerlinkCable, Length=10, Version=1.0.0.3]]
  Supervision = off
  ResponseTimeout = 50
VF-LCR3 : FBE.VF-LCR System (version 04) v04 (OrderNumber=VF-LCR)  [PLK1 -> VF-LCR2.PLK2 (NodeNumber=54) [Cable Type=PowerlinkCable, Length=10, Version=1.0.0.3]; PLK2 -> VF-LCR.PLK1 (NodeNumber=54) [Cable Type=PowerlinkCable, Length=10, Version=1.0.0.3]]
  Supervision = off
  ResponseTimeout = 50
X20AO4622 : X20AO4622 v1.3.0.0  [SS1 -> X20TB12k.SS; SL -> X20BM11h.SL1]
  Supervision = off
  ChannelType03 = 4 to 20mA
X20BM11h : X20BM11 v1.1.0.0  [X2X1 -> X20BM11l.X2X2]
X20BM11k : X20BM11 v1.1.0.0  [X2X1 -> X20BM33a.X2X2]
X20BM11l : X20BM11 v1.1.0.0  [X2X1 -> X20BM11k.X2X2]
X20BM11m : X20BM11 v1.1.0.0  [X2X1 -> X20BM11h.X2X2]
X20BM13a : X20BM13 v1.1.0.0  [X2X1 -> X20BM33c.X2X2]
X20BM33a : X20BM33 v1.1.0.0  [X2X1 -> X20BM13a.X2X2]
X20BM33c : X20BM33 v1.1.0.0  [X2X1 -> 5PC900_TS17_02.IF6]
X20DI9371 : X20DI9371 v1.3.0.0  [SS1 -> X20TB12.SS; SL -> X20BM11k.SL1]
X20DO9322 : X20DO9322 v1.4.0.0  [SS1 -> X20TB12n.SS; SL -> X20BM11l.SL1]
X20DS1119 : X20DS1119 v1.5.0.0  [SS1 -> X20TB12o.SS; SL -> X20BM11m.SL1]
X20SC2432 : X20SC2432 v2.5.0.0  [SS1 -> X20TB52a.SS; SL -> X20BM33a.SL1]
  SafeModuleID = 3
X20SI8110 : X20SI8110 v2.4.0.0  [SS1 -> X20TB52b.SS; SL -> X20BM13a.SL1]
  Supervision = off
X20SLX210 : X20SLX210 v2.4.1.1  [SS1 -> X20TB52f.SS; SL -> X20BM33c.SL1]
  UnsafeOutputUINTs = 8
  UnsafeInputBOOLs = 16
  UnsafeInputUINTs = 8
X20TB12 : X20TB12 v1.0.0.0
X20TB12k : X20TB12 v1.0.0.0
X20TB12n : X20TB12 v1.0.0.0
X20TB12o : X20TB12 v1.0.0.0
X20TB52a : X20TB52 v1.0.0.2
X20TB52b : X20TB52 v1.0.0.2
X20TB52f : X20TB52 v1.0.0.2
```

### Cpu.per - 5PC900_TS17_02/Cpu.per
```iecst
VAR_CONFIG
	gPermConfiguration AT %MB2000; (* *)
	gDataValid AT %MX26000; (* *)
	gPermDataSize AT %MD0; (* *)
END_VAR
```
